KUKA KRL program: f1_Kuka_APT227T02S27.SRC

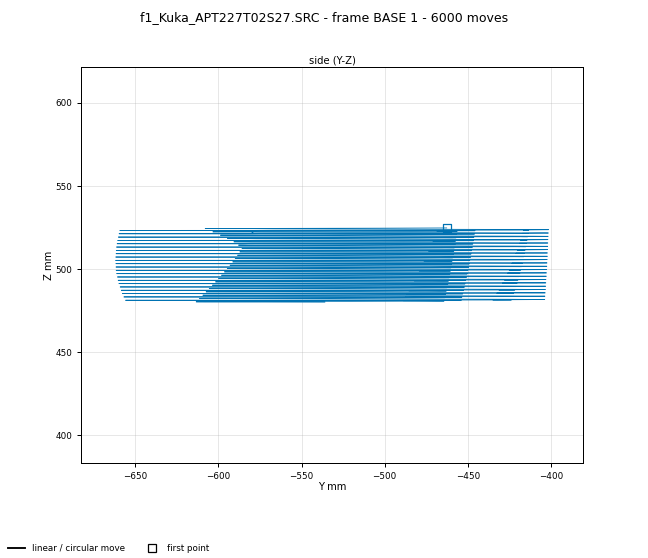
[picture p0: tool path of f1_Kuka_APT227T02S27.SRC in frame BASE 1, 6000 of 6001 moves have a stored position in this frame; points joined in program order, loops and branches not executed]
&ACCESS RVP
&REL 2
&PARAM TEMPLATE = C:\KRC\Roboter\Template\vorgabe
&PARAM EDITMASK = *
DEF f1_Kuka_APT227T02S27()


;FOLD INI;%{PE}%V3.2.0,%MKUKATPBASIS,%CINIT,%VCOMMON,%P
  ;FOLD BAS INI;%{E}%V3.2.0,%MKUKATPBASIS,%CINIT,%VINIT,%P
    GLOBAL INTERRUPT DECL 3 WHEN $STOPMESS==TRUE DO IR_STOPM ( )
    INTERRUPT ON 3
    BAS (#INITMOV,0 )
  ;ENDFOLD (BAS INI)
  ;FOLD USER INI;%{E}%V3.2.0,%MKUKATPUSER,%CINIT,%VINIT,%P
    ;Make your modifications here
  ;ENDFOLD (USER INI)
;ENDFOLD (INI)


;*** Make Null PTP Move
  PTP $pos_act

;*** Auto Load The Correct TOOL Data
  $tool=tool_data[2]

;*** Auto Load The Correct BASE Data
  $base=base_data[1]

  $ADVANCE = 5

;*** Restate Last Velocity
MMPM(30000.0)
SetRPM(8000)
LIN {X -0.077,Y -462.721,Z 524.797,A 0.000,B 0.000,C 90.000,E1 359.484} C_DIS
LIN {X 0.049,Y -465.139,Z 524.785,A 0.000,B 0.000,C 90.000,E1 357.249} C_DIS
LIN {X 0.032,Y -467.419,Z 524.774,A 0.000,B 0.000,C 90.000,E1 355.355} C_DIS
LIN {X 0.101,Y -469.908,Z 524.764,A 0.000,B 0.000,C 90.000,E1 353.457} C_DIS
LIN {X 0.052,Y -472.073,Z 524.755,A 0.000,B 0.000,C 90.000,E1 351.894} C_DIS
LIN {X 0.050,Y -474.231,Z 524.746,A 0.000,B 0.000,C 90.000,E1 350.330} C_DIS
LIN {X 0.160,Y -477.861,Z 524.733,A 0.000,B 0.000,C 90.000,E1 347.825} C_DIS
LIN {X -0.205,Y -484.314,Z 524.712,A 0.000,B 0.000,C 90.000,E1 344.157} C_DIS
LIN {X -0.147,Y -488.007,Z 524.702,A 0.000,B 0.000,C 90.000,E1 342.308} C_DIS
LIN {X 0.164,Y -492.282,Z 524.690,A 0.000,B 0.000,C 90.000,E1 340.134} C_DIS
LIN {X -0.090,Y -495.401,Z 524.681,A 0.000,B 0.000,C 90.000,E1 338.646} C_DIS
LIN {X 0.247,Y -499.060,Z 524.671,A 0.000,B 0.000,C 90.000,E1 336.794} C_DIS
LIN {X -0.055,Y -502.521,Z 524.661,A 0.000,B 0.000,C 90.000,E1 335.025} C_DIS
LIN {X 0.090,Y -505.373,Z 524.653,A 0.000,B 0.000,C 90.000,E1 333.512} C_DIS
LIN {X 0.140,Y -508.743,Z 524.643,A 0.000,B 0.000,C 90.000,E1 331.719} C_DIS
LIN {X -0.036,Y -511.558,Z 524.635,A 0.000,B 0.000,C 90.000,E1 330.255} C_DIS
LIN {X 0.202,Y -514.898,Z 524.625,A 0.000,B 0.000,C 90.000,E1 328.456} C_DIS
LIN {X 0.138,Y -517.811,Z 524.617,A 0.000,B 0.000,C 90.000,E1 326.993} C_DIS
LIN {X -0.035,Y -520.700,Z 524.609,A 0.000,B 0.000,C 90.000,E1 325.548} C_DIS
LIN {X 0.140,Y -523.590,Z 524.601,A 0.000,B 0.000,C 90.000,E1 324.069} C_DIS
LIN {X -0.116,Y -527.585,Z 524.589,A 0.000,B 0.000,C 90.000,E1 322.065} C_DIS
LIN {X 0.087,Y -530.439,Z 524.581,A 0.000,B 0.000,C 90.000,E1 320.598} C_DIS
LIN {X 0.267,Y -533.934,Z 524.572,A 0.000,B 0.000,C 90.000,E1 318.852} C_DIS
LIN {X 0.123,Y -538.133,Z 524.560,A 0.000,B 0.000,C 90.000,E1 316.863} C_DIS
LIN {X 0.048,Y -542.226,Z 524.549,A 0.000,B 0.000,C 90.000,E1 314.879} C_DIS
LIN {X 0.075,Y -546.335,Z 524.538,A 0.000,B 0.000,C 90.000,E1 312.894} C_DIS
LIN {X -0.075,Y -552.002,Z 524.524,A 0.000,B 0.000,C 90.000,E1 310.378} C_DIS
LIN {X -0.188,Y -555.087,Z 524.517,A 0.000,B 0.000,C 90.000,E1 308.991} C_DIS
LIN {X -0.057,Y -556.853,Z 524.512,A 0.000,B 0.000,C 90.000,E1 308.141} C_DIS
LIN {X 0.202,Y -560.643,Z 524.501,A 0.000,B 0.000,C 90.000,E1 306.171} C_DIS
LIN {X -0.099,Y -564.900,Z 524.491,A 0.000,B 0.000,C 90.000,E1 304.405} C_DIS
LIN {X -0.058,Y -566.045,Z 524.489,A 0.000,B 0.000,C 90.000,E1 304.072} C_DIS
LIN {X -0.050,Y -567.206,Z 524.487,A 0.000,B 0.000,C 90.000,E1 303.658} C_DIS
LIN {X -0.322,Y -568.426,Z 524.485,A 0.000,B 0.000,C 90.000,E1 303.372} C_DIS
LIN {X -0.206,Y -569.355,Z 524.484,A 0.000,B 0.000,C 90.000,E1 303.086} C_DIS
LIN {X -0.048,Y -571.821,Z 524.481,A 0.000,B 0.000,C 90.000,E1 302.625} C_DIS
LIN {X 0.075,Y -573.184,Z 524.480,A 0.000,B 0.000,C 90.000,E1 302.339} C_DIS
LIN {X 0.181,Y -575.458,Z 524.478,A 0.000,B 0.000,C 90.000,E1 301.926} C_DIS
LIN {X 0.020,Y -576.825,Z 524.476,A 0.000,B 0.000,C 90.000,E1 301.750} C_DIS
LIN {X 0.006,Y -580.151,Z 524.473,A 0.000,B 0.000,C 90.000,E1 301.209} C_DIS
LIN {X -0.052,Y -584.614,Z 524.470,A 0.000,B 0.000,C 90.000,E1 300.541} C_DIS
LIN {X -0.076,Y -589.187,Z 524.466,A 0.000,B 0.000,C 90.000,E1 299.873} C_DIS
LIN {X 0.186,Y -591.789,Z 524.464,A 0.000,B 0.000,C 90.000,E1 299.461} C_DIS
LIN {X -0.159,Y -597.723,Z 524.459,A 0.000,B 0.000,C 90.000,E1 298.565} C_DIS
LIN {X -0.113,Y -602.317,Z 524.454,A 0.000,B 0.000,C 90.000,E1 297.769} C_DIS
LIN {X -0.182,Y -603.762,Z 524.453,A 0.000,B 0.000,C 90.000,E1 297.513} C_DIS
LIN {X 0.179,Y -606.777,Z 524.448,A 0.000,B 0.000,C 90.000,E1 296.693} C_DIS
LIN {X 0.127,Y -607.269,Z 524.447,A 0.000,B 0.000,C 90.000,E1 296.437} C_DIS
LIN {X 0.031,Y -607.988,Z 524.444,A 0.000,B 0.000,C 90.000,E1 295.924} C_DIS
LIN {X -0.061,Y -607.894,Z 524.441,A 0.000,B 0.000,C 90.000,E1 295.412} C_DIS
LIN {X -0.108,Y -607.568,Z 524.440,A 0.000,B 0.000,C 90.000,E1 295.155} C_DIS
LIN {X -0.202,Y -606.152,Z 524.437,A 0.000,B 0.000,C 90.000,E1 294.643} C_DIS
LIN {X -0.229,Y -605.450,Z 524.436,A 0.000,B 0.000,C 90.000,E1 294.515} C_DIS
LIN {X 0.208,Y -601.708,Z 524.433,A 0.000,B 0.000,C 90.000,E1 293.951} C_DIS
LIN {X 0.191,Y -598.931,Z 524.432,A 0.000,B 0.000,C 90.000,E1 293.695} C_DIS
LIN {X 0.140,Y -595.749,Z 524.430,A 0.000,B 0.000,C 90.000,E1 293.462} C_DIS
LIN {X 0.124,Y -590.658,Z 524.429,A 0.000,B 0.000,C 90.000,E1 293.153} C_DIS
LIN {X -0.082,Y -583.314,Z 524.426,A 0.000,B 0.000,C 90.000,E1 292.717} C_DIS
LIN {X 0.230,Y -582.290,Z 524.426,A 0.000,B 0.000,C 90.000,E1 292.589} C_DIS
LIN {X 0.249,Y -580.640,Z 524.425,A 0.000,B 0.000,C 90.000,E1 292.461} C_DIS
LIN {X 0.267,Y -579.791,Z 524.424,A 0.000,B 0.000,C 90.000,E1 292.333} C_DIS
LIN {X 0.195,Y -579.183,Z 524.424,A 0.000,B 0.000,C 90.000,E1 292.206} C_DIS
LIN {X -0.313,Y -578.283,Z 524.421,A 0.000,B 0.000,C 90.000,E1 291.844} C_DIS
LIN {X -0.004,Y -578.140,Z 524.419,A 0.000,B 0.000,C 90.000,E1 291.408} C_DIS
LIN {X 0.269,Y -578.694,Z 524.410,A 0.000,B 0.000,C 90.000,E1 289.758} C_DIS
LIN {X -0.219,Y -578.876,Z 524.404,A 0.000,B 0.000,C 90.000,E1 288.725} C_DIS
LIN {X 0.047,Y -578.912,Z 524.396,A 0.000,B 0.000,C 90.000,E1 287.347} C_DIS
LIN {X 0.107,Y -578.758,Z 524.390,A 0.000,B 0.000,C 90.000,E1 286.260} C_DIS
LIN {X -0.133,Y -578.314,Z 524.381,A 0.000,B 0.000,C 90.000,E1 284.662} C_DIS
LIN {X -0.250,Y -578.005,Z 524.375,A 0.000,B 0.000,C 90.000,E1 283.592} C_DIS
LIN {X -0.292,Y -577.573,Z 524.368,A 0.000,B 0.000,C 90.000,E1 282.243} C_DIS
LIN {X -0.129,Y -576.982,Z 524.359,A 0.000,B 0.000,C 90.000,E1 280.602} C_DIS
LIN {X -0.094,Y -576.379,Z 524.350,A 0.000,B 0.000,C 90.000,E1 278.973} C_DIS
LIN {X -0.034,Y -575.668,Z 524.339,A 0.000,B 0.000,C 90.000,E1 277.068} C_DIS
LIN {X -0.073,Y -575.376,Z 524.335,A 0.000,B 0.000,C 90.000,E1 276.258} C_DIS
LIN {X 0.152,Y -574.823,Z 524.327,A 0.000,B 0.000,C 90.000,E1 274.878} C_DIS
LIN {X -0.206,Y -574.085,Z 524.320,A 0.000,B 0.000,C 90.000,E1 273.555} C_DIS
LIN {X -0.041,Y -573.161,Z 524.312,A 0.000,B 0.000,C 90.000,E1 272.178} C_DIS
LIN {X 0.244,Y -571.924,Z 524.303,A 0.000,B 0.000,C 90.000,E1 270.516} C_DIS
LIN {X -0.084,Y -570.447,Z 524.294,A 0.000,B 0.000,C 90.000,E1 268.912} C_DIS
LIN {X 0.012,Y -569.173,Z 524.286,A 0.000,B 0.000,C 90.000,E1 267.535} C_DIS
LIN {X -0.033,Y -568.111,Z 524.280,A 0.000,B 0.000,C 90.000,E1 266.445} C_DIS
LIN {X -0.098,Y -567.114,Z 524.274,A 0.000,B 0.000,C 90.000,E1 265.355} C_DIS
LIN {X 0.029,Y -565.712,Z 524.267,A 0.000,B 0.000,C 90.000,E1 263.970} C_DIS
LIN {X -0.019,Y -564.454,Z 524.260,A 0.000,B 0.000,C 90.000,E1 262.875} C_DIS
LIN {X 0.066,Y -562.811,Z 524.253,A 0.000,B 0.000,C 90.000,E1 261.489} C_DIS
LIN {X -0.046,Y -560.309,Z 524.242,A 0.000,B 0.000,C 90.000,E1 259.567} C_DIS
LIN {X 0.183,Y -558.097,Z 524.233,A 0.000,B 0.000,C 90.000,E1 257.881} C_DIS
LIN {X 0.193,Y -556.461,Z 524.227,A 0.000,B 0.000,C 90.000,E1 256.769} C_DIS
LIN {X -0.231,Y -554.729,Z 524.220,A 0.000,B 0.000,C 90.000,E1 255.700} C_DIS
LIN {X -0.021,Y -552.386,Z 524.213,A 0.000,B 0.000,C 90.000,E1 254.283} C_DIS
LIN {X -0.238,Y -549.770,Z 524.205,A 0.000,B 0.000,C 90.000,E1 252.906} C_DIS
LIN {X 0.189,Y -546.847,Z 524.197,A 0.000,B 0.000,C 90.000,E1 251.456} C_DIS
LIN {X -0.198,Y -544.424,Z 524.191,A 0.000,B 0.000,C 90.000,E1 250.369} C_DIS
LIN {X -0.195,Y -541.220,Z 524.183,A 0.000,B 0.000,C 90.000,E1 248.954} C_DIS
LIN {X 0.028,Y -538.498,Z 524.177,A 0.000,B 0.000,C 90.000,E1 247.794} C_DIS
LIN {X -0.085,Y -535.669,Z 524.170,A 0.000,B 0.000,C 90.000,E1 246.666} C_DIS
LIN {X 0.251,Y -532.662,Z 524.164,A 0.000,B 0.000,C 90.000,E1 245.485} C_DIS
LIN {X -0.015,Y -528.732,Z 524.156,A 0.000,B 0.000,C 90.000,E1 244.076} C_DIS
LIN {X -0.035,Y -525.449,Z 524.150,A 0.000,B 0.000,C 90.000,E1 242.922} C_DIS
LIN {X -0.038,Y -520.512,Z 524.140,A 0.000,B 0.000,C 90.000,E1 241.179} C_DIS
LIN {X 0.090,Y -515.420,Z 524.130,A 0.000,B 0.000,C 90.000,E1 239.410} C_DIS
LIN {X -0.068,Y -511.862,Z 524.124,A 0.000,B 0.000,C 90.000,E1 238.250} C_DIS
LIN {X -0.313,Y -506.357,Z 524.114,A 0.000,B 0.000,C 90.000,E1 236.501} C_DIS
LIN {X -0.084,Y -498.136,Z 524.099,A 0.000,B 0.000,C 90.000,E1 233.783} C_DIS
LIN {X -0.034,Y -492.194,Z 524.087,A 0.000,B 0.000,C 90.000,E1 231.662} C_DIS
LIN {X 0.033,Y -487.110,Z 524.077,A 0.000,B 0.000,C 90.000,E1 229.828} C_DIS
LIN {X 0.056,Y -481.384,Z 524.065,A 0.000,B 0.000,C 90.000,E1 227.676} C_DIS
LIN {X 0.112,Y -479.029,Z 524.060,A 0.000,B 0.000,C 90.000,E1 226.743} C_DIS
LIN {X -0.205,Y -474.304,Z 524.049,A 0.000,B 0.000,C 90.000,E1 224.919} C_DIS
LIN {X 0.190,Y -471.260,Z 524.043,A 0.000,B 0.000,C 90.000,E1 223.623} C_DIS
LIN {X 0.039,Y -466.719,Z 524.032,A 0.000,B 0.000,C 90.000,E1 221.757} C_DIS
LIN {X 0.083,Y -463.152,Z 524.023,A 0.000,B 0.000,C 90.000,E1 220.172} C_DIS
LIN {X 0.155,Y -458.881,Z 524.013,A 0.000,B 0.000,C 90.000,E1 218.257} C_DIS
LIN {X 0.118,Y -455.424,Z 524.004,A 0.000,B 0.000,C 90.000,E1 216.664} C_DIS
LIN {X -0.116,Y -450.036,Z 523.990,A 0.000,B 0.000,C 90.000,E1 214.119} C_DIS
LIN {X 0.278,Y -445.614,Z 523.977,A 0.000,B 0.000,C 90.000,E1 211.799} C_DIS
LIN {X 0.084,Y -441.282,Z 523.964,A 0.000,B 0.000,C 90.000,E1 209.539} C_DIS
LIN {X 0.086,Y -438.420,Z 523.955,A 0.000,B 0.000,C 90.000,E1 207.897} C_DIS
LIN {X 0.037,Y -434.989,Z 523.944,A 0.000,B 0.000,C 90.000,E1 205.924} C_DIS
LIN {X 0.124,Y -431.091,Z 523.931,A 0.000,B 0.000,C 90.000,E1 203.590} C_DIS
LIN {X -0.074,Y -426.498,Z 523.914,A 0.000,B 0.000,C 90.000,E1 200.610} C_DIS
LIN {X -0.109,Y -423.681,Z 523.903,A 0.000,B 0.000,C 90.000,E1 198.598} C_DIS
LIN {X 0.106,Y -420.675,Z 523.890,A 0.000,B 0.000,C 90.000,E1 196.205} C_DIS
LIN {X 0.071,Y -418.208,Z 523.879,A 0.000,B 0.000,C 90.000,E1 194.175} C_DIS
LIN {X -0.141,Y -414.972,Z 523.864,A 0.000,B 0.000,C 90.000,E1 191.478} C_DIS
LIN {X 0.201,Y -412.776,Z 523.852,A 0.000,B 0.000,C 90.000,E1 189.378} C_DIS
LIN {X -0.085,Y -410.985,Z 523.843,A 0.000,B 0.000,C 90.000,E1 187.701} C_DIS
LIN {X -0.004,Y -408.416,Z 523.829,A 0.000,B 0.000,C 90.000,E1 185.277} C_DIS
LIN {X -0.157,Y -405.178,Z 523.808,A 0.000,B 0.000,C 90.000,E1 181.489} C_DIS
LIN {X 0.111,Y -404.005,Z 523.799,A 0.000,B 0.000,C 90.000,E1 179.714} C_DIS
LIN {X 0.196,Y -402.337,Z 523.779,A 0.000,B 0.000,C 90.000,E1 176.216} C_DIS
LIN {X -0.068,Y -401.559,Z 523.760,A 0.000,B 0.000,C 90.000,E1 172.761} C_DIS
LIN {X -0.180,Y -401.451,Z 523.746,A 0.000,B 0.000,C 90.000,E1 170.330} C_DIS
LIN {X -0.163,Y -401.675,Z 523.733,A 0.000,B 0.000,C 90.000,E1 167.881} C_DIS
LIN {X 0.118,Y -402.370,Z 523.717,A 0.000,B 0.000,C 90.000,E1 165.046} C_DIS
LIN {X -0.152,Y -403.611,Z 523.700,A 0.000,B 0.000,C 90.000,E1 161.945} C_DIS
LIN {X -0.219,Y -404.872,Z 523.686,A 0.000,B 0.000,C 90.000,E1 159.518} C_DIS
LIN {X -0.062,Y -406.219,Z 523.674,A 0.000,B 0.000,C 90.000,E1 157.411} C_DIS
LIN {X 0.025,Y -407.955,Z 523.661,A 0.000,B 0.000,C 90.000,E1 154.973} C_DIS
LIN {X -0.056,Y -409.262,Z 523.651,A 0.000,B 0.000,C 90.000,E1 153.256} C_DIS
LIN {X 0.148,Y -410.253,Z 523.644,A 0.000,B 0.000,C 90.000,E1 151.847} C_DIS
LIN {X 0.130,Y -411.453,Z 523.634,A 0.000,B 0.000,C 90.000,E1 150.127} C_DIS
LIN {X 0.136,Y -412.492,Z 523.625,A 0.000,B 0.000,C 90.000,E1 148.408} C_DIS
LIN {X 0.023,Y -413.428,Z 523.615,A 0.000,B 0.000,C 90.000,E1 146.707} C_DIS
LIN {X 0.089,Y -414.386,Z 523.604,A 0.000,B 0.000,C 90.000,E1 144.642} C_DIS
LIN {X -0.036,Y -414.932,Z 523.596,A 0.000,B 0.000,C 90.000,E1 143.290} C_DIS
LIN {X -0.080,Y -415.302,Z 523.590,A 0.000,B 0.000,C 90.000,E1 142.271} C_DIS
LIN {X -0.073,Y -415.857,Z 523.581,A 0.000,B 0.000,C 90.000,E1 140.561} C_DIS
LIN {X 0.076,Y -416.211,Z 523.573,A 0.000,B 0.000,C 90.000,E1 139.175} C_DIS
LIN {X -0.127,Y -416.501,Z 523.566,A 0.000,B 0.000,C 90.000,E1 137.838} C_DIS
LIN {X -0.139,Y -416.692,Z 523.556,A 0.000,B 0.000,C 90.000,E1 136.134} C_DIS
LIN {X -0.163,Y -416.692,Z 523.547,A 0.000,B 0.000,C 90.000,E1 134.433} C_DIS
LIN {X -0.067,Y -416.630,Z 523.539,A 0.000,B 0.000,C 90.000,E1 133.056} C_DIS
LIN {X 0.043,Y -416.317,Z 523.532,A 0.000,B 0.000,C 90.000,E1 131.676} C_DIS
LIN {X -0.121,Y -415.764,Z 523.524,A 0.000,B 0.000,C 90.000,E1 130.334} C_DIS
LIN {X -0.028,Y -414.918,Z 523.516,A 0.000,B 0.000,C 90.000,E1 128.955} C_DIS
LIN {X 0.204,Y -413.541,Z 523.505,A 0.000,B 0.000,C 90.000,E1 126.870} C_DIS
LIN {X 0.071,Y -413.402,Z 523.504,A 0.000,B 0.000,C 90.000,E1 126.664} C_DIS
LIN {X 0.032,Y -413.404,Z 523.504,A 0.000,B 0.000,C 90.000,E1 126.664} C_DIS
LIN {X -0.101,Y -415.792,Z 523.499,A 0.000,B 0.000,C 90.000,E1 125.884} C_DIS
LIN {X 0.006,Y -425.244,Z 523.479,A 0.000,B 0.000,C 90.000,E1 122.133} C_DIS
LIN {X -0.061,Y -430.248,Z 523.469,A 0.000,B 0.000,C 90.000,E1 120.463} C_DIS
LIN {X -0.062,Y -431.151,Z 523.467,A 0.000,B 0.000,C 90.000,E1 120.129} C_DIS
LIN {X -0.117,Y -440.260,Z 523.447,A 0.000,B 0.000,C 90.000,E1 116.488} C_DIS
LIN {X 0.076,Y -445.002,Z 523.438,A 0.000,B 0.000,C 90.000,E1 114.823} C_DIS
LIN {X -0.016,Y -453.050,Z 523.419,A 0.000,B 0.000,C 90.000,E1 111.354} C_DIS
LIN {X -0.056,Y -453.112,Z 523.419,A 0.000,B 0.000,C 90.000,E1 111.354} C_DIS
LIN {X 0.157,Y -476.770,Z 523.414,A 0.000,B 0.000,C 90.000,E1 110.482} C_DIS
LIN {X -0.054,Y -494.356,Z 523.410,A 0.000,B 0.000,C 90.000,E1 109.885} C_DIS
LIN {X -0.133,Y -504.552,Z 523.408,A 0.000,B 0.000,C 90.000,E1 109.504} C_DIS
LIN {X -0.077,Y -514.947,Z 523.406,A 0.000,B 0.000,C 90.000,E1 109.087} C_DIS
LIN {X -0.100,Y -526.904,Z 523.403,A 0.000,B 0.000,C 90.000,E1 108.598} C_DIS
LIN {X -0.099,Y -535.317,Z 523.401,A 0.000,B 0.000,C 90.000,E1 108.236} C_DIS
LIN {X -0.030,Y -545.219,Z 523.399,A 0.000,B 0.000,C 90.000,E1 107.764} C_DIS
LIN {X 0.036,Y -552.939,Z 523.396,A 0.000,B 0.000,C 90.000,E1 107.330} C_DIS
LIN {X 0.190,Y -557.612,Z 523.395,A 0.000,B 0.000,C 90.000,E1 107.040} C_DIS
LIN {X -0.112,Y -563.564,Z 523.393,A 0.000,B 0.000,C 90.000,E1 106.677} C_DIS
LIN {X 0.322,Y -567.952,Z 523.391,A 0.000,B 0.000,C 90.000,E1 106.315} C_DIS
LIN {X -0.104,Y -575.047,Z 523.388,A 0.000,B 0.000,C 90.000,E1 105.788} C_DIS
LIN {X -0.054,Y -580.373,Z 523.385,A 0.000,B 0.000,C 90.000,E1 105.300} C_DIS
LIN {X 0.038,Y -585.188,Z 523.382,A 0.000,B 0.000,C 90.000,E1 104.828} C_DIS
LIN {X -0.325,Y -588.649,Z 523.380,A 0.000,B 0.000,C 90.000,E1 104.481} C_DIS
LIN {X 0.157,Y -589.982,Z 523.380,A 0.000,B 0.000,C 90.000,E1 104.300} C_DIS
LIN {X 0.082,Y -595.263,Z 523.376,A 0.000,B 0.000,C 90.000,E1 103.703} C_DIS
LIN {X 0.209,Y -601.269,Z 523.372,A 0.000,B 0.000,C 90.000,E1 102.939} C_DIS
LIN {X 0.282,Y -606.103,Z 523.369,A 0.000,B 0.000,C 90.000,E1 102.299} C_DIS
LIN {X 0.088,Y -611.856,Z 523.364,A 0.000,B 0.000,C 90.000,E1 101.535} C_DIS
LIN {X 0.119,Y -616.974,Z 523.360,A 0.000,B 0.000,C 90.000,E1 100.782} C_DIS
LIN {X -0.141,Y -622.460,Z 523.355,A 0.000,B 0.000,C 90.000,E1 99.905} C_DIS
LIN {X -0.134,Y -626.099,Z 523.351,A 0.000,B 0.000,C 90.000,E1 99.265} C_DIS
LIN {X -0.097,Y -629.550,Z 523.348,A 0.000,B 0.000,C 90.000,E1 98.624} C_DIS
LIN {X -0.154,Y -633.941,Z 523.343,A 0.000,B 0.000,C 90.000,E1 97.757} C_DIS
LIN {X -0.199,Y -637.640,Z 523.339,A 0.000,B 0.000,C 90.000,E1 97.004} C_DIS
LIN {X 0.166,Y -642.290,Z 523.333,A 0.000,B 0.000,C 90.000,E1 95.967} C_DIS
LIN {X 0.129,Y -645.562,Z 523.329,A 0.000,B 0.000,C 90.000,E1 95.220} C_DIS
LIN {X 0.127,Y -648.555,Z 523.325,A 0.000,B 0.000,C 90.000,E1 94.473} C_DIS
LIN {X 0.157,Y -651.236,Z 523.321,A 0.000,B 0.000,C 90.000,E1 93.726} C_DIS
LIN {X -0.059,Y -652.132,Z 523.319,A 0.000,B 0.000,C 90.000,E1 93.498} C_DIS
LIN {X 0.004,Y -654.338,Z 523.315,A 0.000,B 0.000,C 90.000,E1 92.751} C_DIS
LIN {X 0.256,Y -655.673,Z 523.313,A 0.000,B 0.000,C 90.000,E1 92.236} C_DIS
LIN {X -0.115,Y -656.783,Z 523.310,A 0.000,B 0.000,C 90.000,E1 91.776} C_DIS
LIN {X 0.156,Y -657.700,Z 523.307,A 0.000,B 0.000,C 90.000,E1 91.260} C_DIS
LIN {X 0.248,Y -658.652,Z 523.303,A 0.000,B 0.000,C 90.000,E1 90.516} C_DIS
LIN {X -0.122,Y -659.068,Z 523.300,A 0.000,B 0.000,C 90.000,E1 90.057} C_DIS
LIN {X 0.169,Y -659.308,Z 523.298,A 0.000,B 0.000,C 90.000,E1 89.542} C_DIS
LIN {X 0.278,Y -659.279,Z 523.294,A 0.000,B 0.000,C 90.000,E1 88.797} C_DIS
LIN {X -0.091,Y -659.081,Z 523.291,A 0.000,B 0.000,C 90.000,E1 88.339} C_DIS
LIN {X 0.034,Y -658.396,Z 523.287,A 0.000,B 0.000,C 90.000,E1 87.593} C_DIS
LIN {X -0.153,Y -658.166,Z 523.285,A 0.000,B 0.000,C 90.000,E1 87.364} C_DIS
LIN {X -0.030,Y -656.998,Z 523.281,A 0.000,B 0.000,C 90.000,E1 86.617} C_DIS
LIN {X 0.237,Y -656.103,Z 523.279,A 0.000,B 0.000,C 90.000,E1 86.102} C_DIS
LIN {X -0.114,Y -655.018,Z 523.276,A 0.000,B 0.000,C 90.000,E1 85.641} C_DIS
LIN {X -0.020,Y -653.077,Z 523.272,A 0.000,B 0.000,C 90.000,E1 84.894} C_DIS
LIN {X -0.101,Y -650.007,Z 523.266,A 0.000,B 0.000,C 90.000,E1 83.913} C_DIS
LIN {X -0.062,Y -647.376,Z 523.262,A 0.000,B 0.000,C 90.000,E1 83.166} C_DIS
LIN {X -0.219,Y -643.396,Z 523.257,A 0.000,B 0.000,C 90.000,E1 82.186} C_DIS
LIN {X -0.170,Y -640.058,Z 523.252,A 0.000,B 0.000,C 90.000,E1 81.432} C_DIS
LIN {X -0.015,Y -637.052,Z 523.249,A 0.000,B 0.000,C 90.000,E1 80.792} C_DIS
LIN {X 0.114,Y -633.781,Z 523.245,A 0.000,B 0.000,C 90.000,E1 80.151} C_DIS
LIN {X -0.096,Y -628.841,Z 523.240,A 0.000,B 0.000,C 90.000,E1 79.285} C_DIS
LIN {X 0.283,Y -626.571,Z 523.238,A 0.000,B 0.000,C 90.000,E1 78.870} C_DIS
LIN {X 0.148,Y -621.784,Z 523.234,A 0.000,B 0.000,C 90.000,E1 78.117} C_DIS
LIN {X -0.289,Y -618.585,Z 523.231,A 0.000,B 0.000,C 90.000,E1 77.645} C_DIS
LIN {X 0.137,Y -613.548,Z 523.227,A 0.000,B 0.000,C 90.000,E1 76.881} C_DIS
LIN {X 0.135,Y -607.509,Z 523.223,A 0.000,B 0.000,C 90.000,E1 76.117} C_DIS
LIN {X 0.201,Y -602.910,Z 523.220,A 0.000,B 0.000,C 90.000,E1 75.589} C_DIS
LIN {X -0.023,Y -598.092,Z 523.217,A 0.000,B 0.000,C 90.000,E1 75.102} C_DIS
LIN {X -0.254,Y -591.907,Z 523.214,A 0.000,B 0.000,C 90.000,E1 74.519} C_DIS
LIN {X 0.284,Y -586.401,Z 523.211,A 0.000,B 0.000,C 90.000,E1 73.976} C_DIS
LIN {X -0.192,Y -580.627,Z 523.209,A 0.000,B 0.000,C 90.000,E1 73.559} C_DIS
LIN {X -0.270,Y -574.898,Z 523.206,A 0.000,B 0.000,C 90.000,E1 73.142} C_DIS
LIN {X 0.184,Y -570.285,Z 523.204,A 0.000,B 0.000,C 90.000,E1 72.779} C_DIS
LIN {X 0.244,Y -563.718,Z 523.202,A 0.000,B 0.000,C 90.000,E1 72.362} C_DIS
LIN {X -0.177,Y -558.688,Z 523.201,A 0.000,B 0.000,C 90.000,E1 72.127} C_DIS
LIN {X -0.186,Y -553.667,Z 523.199,A 0.000,B 0.000,C 90.000,E1 71.873} C_DIS
LIN {X 0.090,Y -546.412,Z 523.198,A 0.000,B 0.000,C 90.000,E1 71.529} C_DIS
LIN {X -0.015,Y -540.962,Z 523.196,A 0.000,B 0.000,C 90.000,E1 71.329} C_DIS
LIN {X -0.084,Y -535.612,Z 523.195,A 0.000,B 0.000,C 90.000,E1 71.148} C_DIS
LIN {X 0.021,Y -527.801,Z 523.194,A 0.000,B 0.000,C 90.000,E1 70.913} C_DIS
LIN {X -0.208,Y -514.834,Z 523.192,A 0.000,B 0.000,C 90.000,E1 70.604} C_DIS
LIN {X 0.078,Y -503.831,Z 523.191,A 0.000,B 0.000,C 90.000,E1 70.315} C_DIS
LIN {X 0.160,Y -494.116,Z 523.190,A 0.000,B 0.000,C 90.000,E1 70.115} C_DIS
LIN {X -0.070,Y -483.073,Z 523.189,A 0.000,B 0.000,C 90.000,E1 69.934} C_DIS
LIN {X -0.068,Y -469.667,Z 523.187,A 0.000,B 0.000,C 90.000,E1 69.699} C_DIS
LIN {X -0.102,Y -469.642,Z 523.187,A 0.000,B 0.000,C 90.000,E1 69.699} C_DIS
LIN {X -0.100,Y -465.762,Z 523.173,A 0.000,B 0.000,C 90.000,E1 67.155} C_DIS
LIN {X 0.144,Y -463.664,Z 523.168,A 0.000,B 0.000,C 90.000,E1 66.177} C_DIS
LIN {X 0.230,Y -455.727,Z 523.145,A 0.000,B 0.000,C 90.000,E1 62.025} C_DIS
LIN {X 0.119,Y -455.083,Z 523.143,A 0.000,B 0.000,C 90.000,E1 61.719} C_DIS
LIN {X -0.054,Y -446.436,Z 523.122,A 0.000,B 0.000,C 90.000,E1 57.867} C_DIS
LIN {X 0.076,Y -445.686,Z 523.119,A 0.000,B 0.000,C 90.000,E1 57.454} C_DIS
LIN {X 0.036,Y -445.699,Z 523.119,A 0.000,B 0.000,C 90.000,E1 57.454} C_DIS
LIN {X 0.223,Y -450.097,Z 523.111,A 0.000,B 0.000,C 90.000,E1 55.881} C_DIS
LIN {X -0.288,Y -452.595,Z 523.105,A 0.000,B 0.000,C 90.000,E1 54.975} C_DIS
LIN {X -0.060,Y -456.379,Z 523.096,A 0.000,B 0.000,C 90.000,E1 53.336} C_DIS
LIN {X 0.037,Y -457.767,Z 523.093,A 0.000,B 0.000,C 90.000,E1 52.683} C_DIS
LIN {X -0.118,Y -459.541,Z 523.087,A 0.000,B 0.000,C 90.000,E1 51.743} C_DIS
LIN {X -0.127,Y -462.114,Z 523.079,A 0.000,B 0.000,C 90.000,E1 50.150} C_DIS
LIN {X 0.102,Y -463.873,Z 523.072,A 0.000,B 0.000,C 90.000,E1 48.852} C_DIS
LIN {X -0.044,Y -465.024,Z 523.066,A 0.000,B 0.000,C 90.000,E1 47.919} C_DIS
LIN {X -0.174,Y -466.013,Z 523.061,A 0.000,B 0.000,C 90.000,E1 46.986} C_DIS
LIN {X -0.295,Y -466.818,Z 523.056,A 0.000,B 0.000,C 90.000,E1 46.053} C_DIS
LIN {X -0.084,Y -467.481,Z 523.050,A 0.000,B 0.000,C 90.000,E1 45.081} C_DIS
LIN {X 0.137,Y -468.036,Z 523.045,A 0.000,B 0.000,C 90.000,E1 44.109} C_DIS
LIN {X 0.114,Y -468.446,Z 523.038,A 0.000,B 0.000,C 90.000,E1 42.852} C_DIS
LIN {X 0.095,Y -468.615,Z 523.031,A 0.000,B 0.000,C 90.000,E1 41.595} C_DIS
LIN {X 0.119,Y -468.463,Z 523.024,A 0.000,B 0.000,C 90.000,E1 40.334} C_DIS
LIN {X -0.216,Y -468.162,Z 523.017,A 0.000,B 0.000,C 90.000,E1 39.116} C_DIS
LIN {X -0.016,Y -467.483,Z 523.007,A 0.000,B 0.000,C 90.000,E1 37.202} C_DIS
LIN {X 0.215,Y -466.709,Z 522.998,A 0.000,B 0.000,C 90.000,E1 35.598} C_DIS
LIN {X 0.051,Y -465.881,Z 522.989,A 0.000,B 0.000,C 90.000,E1 34.040} C_DIS
LIN {X -0.007,Y -464.940,Z 522.980,A 0.000,B 0.000,C 90.000,E1 32.467} C_DIS
LIN {X 0.068,Y -464.002,Z 522.972,A 0.000,B 0.000,C 90.000,E1 30.875} C_DIS
LIN {X -0.138,Y -462.740,Z 522.961,A 0.000,B 0.000,C 90.000,E1 28.999} C_DIS
LIN {X -0.010,Y -461.464,Z 522.951,A 0.000,B 0.000,C 90.000,E1 27.078} C_DIS
LIN {X 0.014,Y -460.040,Z 522.938,A 0.000,B 0.000,C 90.000,E1 24.847} C_DIS
LIN {X -0.114,Y -459.033,Z 522.927,A 0.000,B 0.000,C 90.000,E1 22.950} C_DIS
LIN {X 0.050,Y -457.942,Z 522.913,A 0.000,B 0.000,C 90.000,E1 20.375} C_DIS
LIN {X -0.070,Y -457.267,Z 522.903,A 0.000,B 0.000,C 90.000,E1 18.471} C_DIS
LIN {X -0.208,Y -456.570,Z 522.887,A 0.000,B 0.000,C 90.000,E1 15.607} C_DIS
LIN {X -0.045,Y -456.427,Z 522.871,A 0.000,B 0.000,C 90.000,E1 12.703} C_DIS
LIN {X -0.056,Y -456.664,Z 522.860,A 0.000,B 0.000,C 90.000,E1 10.782} C_DIS
LIN {X 0.175,Y -457.228,Z 522.847,A 0.000,B 0.000,C 90.000,E1 8.511} C_DIS
LIN {X -0.173,Y -458.085,Z 522.835,A 0.000,B 0.000,C 90.000,E1 6.315} C_DIS
LIN {X 0.090,Y -459.503,Z 522.821,A 0.000,B 0.000,C 90.000,E1 3.726} C_DIS
LIN {X 0.138,Y -461.050,Z 522.808,A 0.000,B 0.000,C 90.000,E1 1.489} C_DIS
LIN {X -0.076,Y -462.867,Z 522.797,A 0.000,B 0.000,C 90.000,E1 359.484} C_DIS
LIN {X 0.054,Y -465.273,Z 522.785,A 0.000,B 0.000,C 90.000,E1 357.249} C_DIS
LIN {X 0.039,Y -467.544,Z 522.774,A 0.000,B 0.000,C 90.000,E1 355.355} C_DIS
LIN {X 0.111,Y -470.032,Z 522.764,A 0.000,B 0.000,C 90.000,E1 353.457} C_DIS
LIN {X -0.111,Y -472.621,Z 522.753,A 0.000,B 0.000,C 90.000,E1 351.602} C_DIS
LIN {X -0.103,Y -474.769,Z 522.745,A 0.000,B 0.000,C 90.000,E1 350.038} C_DIS
LIN {X 0.178,Y -477.984,Z 522.733,A 0.000,B 0.000,C 90.000,E1 347.825} C_DIS
LIN {X -0.041,Y -483.873,Z 522.714,A 0.000,B 0.000,C 90.000,E1 344.448} C_DIS
LIN {X -0.119,Y -488.161,Z 522.702,A 0.000,B 0.000,C 90.000,E1 342.308} C_DIS
LIN {X -0.264,Y -492.468,Z 522.690,A 0.000,B 0.000,C 90.000,E1 340.188} C_DIS
LIN {X -0.053,Y -495.579,Z 522.681,A 0.000,B 0.000,C 90.000,E1 338.646} C_DIS
LIN {X 0.226,Y -498.641,Z 522.673,A 0.000,B 0.000,C 90.000,E1 337.102} C_DIS
LIN {X 0.095,Y -501.572,Z 522.665,A 0.000,B 0.000,C 90.000,E1 335.613} C_DIS
LIN {X -0.237,Y -504.462,Z 522.656,A 0.000,B 0.000,C 90.000,E1 334.152} C_DIS
LIN {X -0.207,Y -507.868,Z 522.646,A 0.000,B 0.000,C 90.000,E1 332.359} C_DIS
LIN {X 0.131,Y -511.238,Z 522.636,A 0.000,B 0.000,C 90.000,E1 330.539} C_DIS
LIN {X -0.085,Y -514.653,Z 522.627,A 0.000,B 0.000,C 90.000,E1 328.791} C_DIS
LIN {X -0.223,Y -518.145,Z 522.617,A 0.000,B 0.000,C 90.000,E1 327.041} C_DIS
LIN {X 0.045,Y -521.037,Z 522.609,A 0.000,B 0.000,C 90.000,E1 325.548} C_DIS
LIN {X -0.197,Y -523.951,Z 522.601,A 0.000,B 0.000,C 90.000,E1 324.116} C_DIS
LIN {X 0.011,Y -527.420,Z 522.591,A 0.000,B 0.000,C 90.000,E1 322.351} C_DIS
LIN {X 0.213,Y -530.322,Z 522.583,A 0.000,B 0.000,C 90.000,E1 320.884} C_DIS
LIN {X 0.046,Y -533.791,Z 522.573,A 0.000,B 0.000,C 90.000,E1 319.175} C_DIS
LIN {X -0.093,Y -536.764,Z 522.565,A 0.000,B 0.000,C 90.000,E1 317.757} C_DIS
LIN {X -0.145,Y -539.195,Z 522.559,A 0.000,B 0.000,C 90.000,E1 316.620} C_DIS
LIN {X 0.191,Y -543.256,Z 522.548,A 0.000,B 0.000,C 90.000,E1 314.595} C_DIS
LIN {X -0.143,Y -546.692,Z 522.539,A 0.000,B 0.000,C 90.000,E1 312.933} C_DIS
LIN {X 0.091,Y -552.259,Z 522.524,A 0.000,B 0.000,C 90.000,E1 310.378} C_DIS
LIN {X -0.086,Y -554.742,Z 522.518,A 0.000,B 0.000,C 90.000,E1 309.277} C_DIS
LIN {X -0.225,Y -557.133,Z 522.512,A 0.000,B 0.000,C 90.000,E1 308.177} C_DIS
LIN {X 0.110,Y -559.275,Z 522.506,A 0.000,B 0.000,C 90.000,E1 307.030} C_DIS
LIN {X -0.016,Y -565.229,Z 522.490,A 0.000,B 0.000,C 90.000,E1 304.278} C_DIS
LIN {X 0.202,Y -566.732,Z 522.487,A 0.000,B 0.000,C 90.000,E1 303.706} C_DIS
LIN {X -0.001,Y -567.396,Z 522.486,A 0.000,B 0.000,C 90.000,E1 303.452} C_DIS
LIN {X 0.228,Y -569.107,Z 522.483,A 0.000,B 0.000,C 90.000,E1 302.880} C_DIS
LIN {X -0.011,Y -569.952,Z 522.482,A 0.000,B 0.000,C 90.000,E1 302.752} C_DIS
LIN {X 0.109,Y -571.087,Z 522.480,A 0.000,B 0.000,C 90.000,E1 302.467} C_DIS
LIN {X -0.076,Y -572.006,Z 522.479,A 0.000,B 0.000,C 90.000,E1 302.212} C_DIS
LIN {X 0.049,Y -573.384,Z 522.477,A 0.000,B 0.000,C 90.000,E1 301.926} C_DIS
LIN {X -0.038,Y -573.976,Z 522.477,A 0.000,B 0.000,C 90.000,E1 301.799} C_DIS
LIN {X -0.073,Y -576.985,Z 522.474,A 0.000,B 0.000,C 90.000,E1 301.258} C_DIS
LIN {X -0.014,Y -579.173,Z 522.471,A 0.000,B 0.000,C 90.000,E1 300.846} C_DIS
LIN {X 0.320,Y -588.155,Z 522.463,A 0.000,B 0.000,C 90.000,E1 299.333} C_DIS
LIN {X 0.121,Y -595.328,Z 522.457,A 0.000,B 0.000,C 90.000,E1 298.153} C_DIS
LIN {X -0.015,Y -597.485,Z 522.454,A 0.000,B 0.000,C 90.000,E1 297.769} C_DIS
LIN {X -0.220,Y -600.522,Z 522.451,A 0.000,B 0.000,C 90.000,E1 297.129} C_DIS
LIN {X -0.295,Y -601.462,Z 522.449,A 0.000,B 0.000,C 90.000,E1 296.873} C_DIS
LIN {X 0.106,Y -602.721,Z 522.446,A 0.000,B 0.000,C 90.000,E1 296.309} C_DIS
LIN {X 0.041,Y -603.162,Z 522.445,A 0.000,B 0.000,C 90.000,E1 296.052} C_DIS
LIN {X -0.022,Y -603.349,Z 522.443,A 0.000,B 0.000,C 90.000,E1 295.796} C_DIS
LIN {X -0.083,Y -603.390,Z 522.442,A 0.000,B 0.000,C 90.000,E1 295.540} C_DIS
LIN {X -0.205,Y -602.726,Z 522.439,A 0.000,B 0.000,C 90.000,E1 295.027} C_DIS
LIN {X -0.269,Y -602.259,Z 522.438,A 0.000,B 0.000,C 90.000,E1 294.771} C_DIS
LIN {X -0.301,Y -601.402,Z 522.437,A 0.000,B 0.000,C 90.000,E1 294.643} C_DIS
LIN {X 0.143,Y -599.371,Z 522.435,A 0.000,B 0.000,C 90.000,E1 294.207} C_DIS
LIN {X 0.107,Y -598.411,Z 522.434,A 0.000,B 0.000,C 90.000,E1 294.079} C_DIS
LIN {X 0.100,Y -594.628,Z 522.432,A 0.000,B 0.000,C 90.000,E1 293.695} C_DIS
LIN {X -0.225,Y -592.255,Z 522.431,A 0.000,B 0.000,C 90.000,E1 293.515} C_DIS
LIN {X 0.155,Y -587.306,Z 522.429,A 0.000,B 0.000,C 90.000,E1 293.131} C_DIS
LIN {X -0.058,Y -583.478,Z 522.427,A 0.000,B 0.000,C 90.000,E1 292.898} C_DIS
LIN {X -0.013,Y -581.170,Z 522.426,A 0.000,B 0.000,C 90.000,E1 292.642} C_DIS
LIN {X -0.228,Y -580.119,Z 522.425,A 0.000,B 0.000,C 90.000,E1 292.461} C_DIS
LIN {X -0.298,Y -579.673,Z 522.424,A 0.000,B 0.000,C 90.000,E1 292.333} C_DIS
LIN {X -0.135,Y -579.246,Z 522.422,A 0.000,B 0.000,C 90.000,E1 291.972} C_DIS
LIN {X 0.105,Y -579.080,Z 522.419,A 0.000,B 0.000,C 90.000,E1 291.408} C_DIS
LIN {X -0.146,Y -579.694,Z 522.410,A 0.000,B 0.000,C 90.000,E1 289.812} C_DIS
LIN {X -0.076,Y -579.922,Z 522.404,A 0.000,B 0.000,C 90.000,E1 288.725} C_DIS
LIN {X -0.344,Y -579.978,Z 522.397,A 0.000,B 0.000,C 90.000,E1 287.402} C_DIS
LIN {X 0.284,Y -579.845,Z 522.391,A 0.000,B 0.000,C 90.000,E1 286.260} C_DIS
LIN {X -0.152,Y -579.513,Z 522.383,A 0.000,B 0.000,C 90.000,E1 284.954} C_DIS
LIN {X -0.034,Y -579.170,Z 522.376,A 0.000,B 0.000,C 90.000,E1 283.592} C_DIS
LIN {X 0.164,Y -578.705,Z 522.367,A 0.000,B 0.000,C 90.000,E1 281.951} C_DIS
LIN {X -0.002,Y -578.040,Z 522.356,A 0.000,B 0.000,C 90.000,E1 280.074} C_DIS
LIN {X -0.253,Y -577.566,Z 522.349,A 0.000,B 0.000,C 90.000,E1 278.746} C_DIS
LIN {X -0.082,Y -576.922,Z 522.338,A 0.000,B 0.000,C 90.000,E1 276.834} C_DIS
LIN {X -0.209,Y -576.256,Z 522.329,A 0.000,B 0.000,C 90.000,E1 275.220} C_DIS
LIN {X 0.026,Y -575.531,Z 522.321,A 0.000,B 0.000,C 90.000,E1 273.841} C_DIS
LIN {X 0.213,Y -574.618,Z 522.314,A 0.000,B 0.000,C 90.000,E1 272.465} C_DIS
LIN {X -0.046,Y -573.364,Z 522.305,A 0.000,B 0.000,C 90.000,E1 270.859} C_DIS
LIN {X -0.049,Y -572.382,Z 522.299,A 0.000,B 0.000,C 90.000,E1 269.771} C_DIS
LIN {X 0.065,Y -571.127,Z 522.291,A 0.000,B 0.000,C 90.000,E1 268.396} C_DIS
LIN {X -0.242,Y -569.545,Z 522.282,A 0.000,B 0.000,C 90.000,E1 266.788} C_DIS
LIN {X -0.164,Y -568.194,Z 522.274,A 0.000,B 0.000,C 90.000,E1 265.412} C_DIS
LIN {X -0.076,Y -566.738,Z 522.267,A 0.000,B 0.000,C 90.000,E1 264.033} C_DIS
LIN {X -0.049,Y -565.480,Z 522.261,A 0.000,B 0.000,C 90.000,E1 262.932} C_DIS
LIN {X 0.055,Y -563.711,Z 522.253,A 0.000,B 0.000,C 90.000,E1 261.546} C_DIS
LIN {X -0.188,Y -561.533,Z 522.244,A 0.000,B 0.000,C 90.000,E1 259.916} C_DIS
LIN {X -0.075,Y -559.691,Z 522.236,A 0.000,B 0.000,C 90.000,E1 258.522} C_DIS
LIN {X -0.037,Y -558.114,Z 522.230,A 0.000,B 0.000,C 90.000,E1 257.409} C_DIS
LIN {X 0.239,Y -555.963,Z 522.222,A 0.000,B 0.000,C 90.000,E1 255.992} C_DIS
LIN {X -0.058,Y -553.636,Z 522.215,A 0.000,B 0.000,C 90.000,E1 254.629} C_DIS
LIN {X 0.019,Y -551.595,Z 522.208,A 0.000,B 0.000,C 90.000,E1 253.504} C_DIS
LIN {X -0.041,Y -549.931,Z 522.204,A 0.000,B 0.000,C 90.000,E1 252.670} C_DIS
LIN {X -0.133,Y -546.954,Z 522.196,A 0.000,B 0.000,C 90.000,E1 251.275} C_DIS
LIN {X 0.179,Y -544.489,Z 522.190,A 0.000,B 0.000,C 90.000,E1 250.115} C_DIS
LIN {X -0.245,Y -541.875,Z 522.183,A 0.000,B 0.000,C 90.000,E1 249.028} C_DIS
LIN {X 0.185,Y -539.133,Z 522.177,A 0.000,B 0.000,C 90.000,E1 247.847} C_DIS
LIN {X -0.127,Y -536.284,Z 522.171,A 0.000,B 0.000,C 90.000,E1 246.741} C_DIS
LIN {X 0.149,Y -532.493,Z 522.163,A 0.000,B 0.000,C 90.000,E1 245.281} C_DIS
LIN {X 0.130,Y -528.487,Z 522.155,A 0.000,B 0.000,C 90.000,E1 243.845} C_DIS
LIN {X 0.028,Y -524.363,Z 522.147,A 0.000,B 0.000,C 90.000,E1 242.410} C_DIS
LIN {X -0.134,Y -520.168,Z 522.139,A 0.000,B 0.000,C 90.000,E1 240.973} C_DIS
LIN {X 0.069,Y -515.913,Z 522.131,A 0.000,B 0.000,C 90.000,E1 239.488} C_DIS
LIN {X -0.084,Y -512.372,Z 522.124,A 0.000,B 0.000,C 90.000,E1 238.329} C_DIS
LIN {X -0.045,Y -506.820,Z 522.114,A 0.000,B 0.000,C 90.000,E1 236.548} C_DIS
LIN {X 0.039,Y -499.410,Z 522.101,A 0.000,B 0.000,C 90.000,E1 234.149} C_DIS
LIN {X -0.029,Y -492.535,Z 522.087,A 0.000,B 0.000,C 90.000,E1 231.743} C_DIS
LIN {X 0.043,Y -487.478,Z 522.077,A 0.000,B 0.000,C 90.000,E1 229.908} C_DIS
LIN {X -0.060,Y -482.513,Z 522.067,A 0.000,B 0.000,C 90.000,E1 228.081} C_DIS
LIN {X 0.134,Y -479.374,Z 522.060,A 0.000,B 0.000,C 90.000,E1 226.824} C_DIS
LIN {X -0.175,Y -474.633,Z 522.050,A 0.000,B 0.000,C 90.000,E1 225.000} C_DIS
LIN {X 0.223,Y -471.574,Z 522.043,A 0.000,B 0.000,C 90.000,E1 223.704} C_DIS
LIN {X 0.148,Y -466.265,Z 522.031,A 0.000,B 0.000,C 90.000,E1 221.515} C_DIS
LIN {X 0.130,Y -463.428,Z 522.024,A 0.000,B 0.000,C 90.000,E1 220.253} C_DIS
LIN {X -0.150,Y -459.155,Z 522.013,A 0.000,B 0.000,C 90.000,E1 218.382} C_DIS
LIN {X -0.185,Y -455.701,Z 522.004,A 0.000,B 0.000,C 90.000,E1 216.790} C_DIS
LIN {X -0.126,Y -450.986,Z 521.992,A 0.000,B 0.000,C 90.000,E1 214.532} C_DIS
LIN {X -0.013,Y -445.880,Z 521.977,A 0.000,B 0.000,C 90.000,E1 211.926} C_DIS
LIN {X -0.199,Y -441.572,Z 521.965,A 0.000,B 0.000,C 90.000,E1 209.667} C_DIS
LIN {X 0.196,Y -438.684,Z 521.956,A 0.000,B 0.000,C 90.000,E1 207.975} C_DIS
LIN {X -0.042,Y -435.245,Z 521.945,A 0.000,B 0.000,C 90.000,E1 206.027} C_DIS
LIN {X 0.046,Y -431.902,Z 521.934,A 0.000,B 0.000,C 90.000,E1 204.027} C_DIS
LIN {X 0.074,Y -427.660,Z 521.919,A 0.000,B 0.000,C 90.000,E1 201.354} C_DIS
LIN {X -0.131,Y -424.348,Z 521.906,A 0.000,B 0.000,C 90.000,E1 199.033} C_DIS
LIN {X 0.005,Y -420.834,Z 521.891,A 0.000,B 0.000,C 90.000,E1 196.315} C_DIS
LIN {X 0.213,Y -418.764,Z 521.881,A 0.000,B 0.000,C 90.000,E1 194.592} C_DIS
LIN {X 0.127,Y -417.108,Z 521.874,A 0.000,B 0.000,C 90.000,E1 193.244} C_DIS
LIN {X -0.154,Y -414.379,Z 521.860,A 0.000,B 0.000,C 90.000,E1 190.894} C_DIS
LIN {X 0.025,Y -412.948,Z 521.853,A 0.000,B 0.000,C 90.000,E1 189.500} C_DIS
LIN {X 0.214,Y -411.159,Z 521.843,A 0.000,B 0.000,C 90.000,E1 187.757} C_DIS
LIN {X -0.151,Y -409.332,Z 521.834,A 0.000,B 0.000,C 90.000,E1 186.087} C_DIS
LIN {X 0.147,Y -405.312,Z 521.809,A 0.000,B 0.000,C 90.000,E1 181.547} C_DIS
LIN {X -0.017,Y -403.930,Z 521.797,A 0.000,B 0.000,C 90.000,E1 179.484} C_DIS
LIN {X 0.063,Y -402.304,Z 521.778,A 0.000,B 0.000,C 90.000,E1 175.988} C_DIS
LIN {X -0.150,Y -401.653,Z 521.760,A 0.000,B 0.000,C 90.000,E1 172.875} C_DIS
LIN {X 0.134,Y -401.581,Z 521.745,A 0.000,B 0.000,C 90.000,E1 170.038} C_DIS
LIN {X -0.170,Y -401.976,Z 521.727,A 0.000,B 0.000,C 90.000,E1 166.937} C_DIS
LIN {X 0.140,Y -402.682,Z 521.714,A 0.000,B 0.000,C 90.000,E1 164.448} C_DIS
LIN {X -0.092,Y -403.880,Z 521.698,A 0.000,B 0.000,C 90.000,E1 161.692} C_DIS
LIN {X -0.038,Y -405.408,Z 521.683,A 0.000,B 0.000,C 90.000,E1 158.901} C_DIS
LIN {X 0.134,Y -406.756,Z 521.671,A 0.000,B 0.000,C 90.000,E1 156.794} C_DIS
LIN {X 0.130,Y -408.323,Z 521.660,A 0.000,B 0.000,C 90.000,E1 154.717} C_DIS
LIN {X 0.057,Y -409.667,Z 521.650,A 0.000,B 0.000,C 90.000,E1 152.999} C_DIS
LIN {X -0.093,Y -410.650,Z 521.642,A 0.000,B 0.000,C 90.000,E1 151.641} C_DIS
LIN {X -0.030,Y -411.645,Z 521.635,A 0.000,B 0.000,C 90.000,E1 150.255} C_DIS
LIN {X -0.018,Y -412.720,Z 521.625,A 0.000,B 0.000,C 90.000,E1 148.535} C_DIS
LIN {X -0.124,Y -413.667,Z 521.616,A 0.000,B 0.000,C 90.000,E1 146.834} C_DIS
LIN {X -0.047,Y -414.678,Z 521.604,A 0.000,B 0.000,C 90.000,E1 144.769} C_DIS
LIN {X -0.165,Y -415.283,Z 521.597,A 0.000,B 0.000,C 90.000,E1 143.417} C_DIS
LIN {X 0.128,Y -415.687,Z 521.591,A 0.000,B 0.000,C 90.000,E1 142.351} C_DIS
LIN {X 0.140,Y -416.272,Z 521.581,A 0.000,B 0.000,C 90.000,E1 140.642} C_DIS
LIN {X -0.019,Y -416.660,Z 521.574,A 0.000,B 0.000,C 90.000,E1 139.299} C_DIS
LIN {X 0.099,Y -416.955,Z 521.566,A 0.000,B 0.000,C 90.000,E1 137.919} C_DIS
LIN {X 0.096,Y -417.205,Z 521.557,A 0.000,B 0.000,C 90.000,E1 136.215} C_DIS
LIN {X 0.082,Y -417.197,Z 521.547,A 0.000,B 0.000,C 90.000,E1 134.514} C_DIS
LIN {X -0.100,Y -417.119,Z 521.540,A 0.000,B 0.000,C 90.000,E1 133.176} C_DIS
LIN {X 0.120,Y -416.910,Z 521.534,A 0.000,B 0.000,C 90.000,E1 132.123} C_DIS
LIN {X -0.224,Y -416.579,Z 521.529,A 0.000,B 0.000,C 90.000,E1 131.148} C_DIS
LIN {X 0.019,Y -416.043,Z 521.523,A 0.000,B 0.000,C 90.000,E1 130.092} C_DIS
LIN {X 0.032,Y -414.910,Z 521.513,A 0.000,B 0.000,C 90.000,E1 128.382} C_DIS
LIN {X -0.062,Y -413.700,Z 521.503,A 0.000,B 0.000,C 90.000,E1 126.583} C_DIS
LIN {X -0.101,Y -413.700,Z 521.503,A 0.000,B 0.000,C 90.000,E1 126.583} C_DIS
LIN {X -0.138,Y -415.472,Z 521.500,A 0.000,B 0.000,C 90.000,E1 126.011} C_DIS
LIN {X -0.079,Y -425.866,Z 521.477,A 0.000,B 0.000,C 90.000,E1 121.926} C_DIS
LIN {X -0.135,Y -430.888,Z 521.468,A 0.000,B 0.000,C 90.000,E1 120.256} C_DIS
LIN {X -0.206,Y -439.935,Z 521.448,A 0.000,B 0.000,C 90.000,E1 116.616} C_DIS
LIN {X -0.020,Y -444.728,Z 521.439,A 0.000,B 0.000,C 90.000,E1 114.951} C_DIS
LIN {X -0.108,Y -453.892,Z 521.417,A 0.000,B 0.000,C 90.000,E1 111.046} C_DIS
LIN {X -0.141,Y -453.972,Z 521.417,A 0.000,B 0.000,C 90.000,E1 111.046} C_DIS
LIN {X -0.058,Y -480.080,Z 521.412,A 0.000,B 0.000,C 90.000,E1 110.120} C_DIS
LIN {X -0.046,Y -494.081,Z 521.409,A 0.000,B 0.000,C 90.000,E1 109.631} C_DIS
LIN {X -0.196,Y -500.934,Z 521.408,A 0.000,B 0.000,C 90.000,E1 109.396} C_DIS
LIN {X -0.204,Y -518.233,Z 521.404,A 0.000,B 0.000,C 90.000,E1 108.725} C_DIS
LIN {X -0.038,Y -528.484,Z 521.402,A 0.000,B 0.000,C 90.000,E1 108.290} C_DIS
LIN {X 0.009,Y -535.181,Z 521.400,A 0.000,B 0.000,C 90.000,E1 108.000} C_DIS
LIN {X 0.133,Y -545.096,Z 521.398,A 0.000,B 0.000,C 90.000,E1 107.528} C_DIS
LIN {X -0.154,Y -551.374,Z 521.396,A 0.000,B 0.000,C 90.000,E1 107.221} C_DIS
LIN {X 0.161,Y -558.900,Z 521.393,A 0.000,B 0.000,C 90.000,E1 106.749} C_DIS
LIN {X -0.174,Y -563.341,Z 521.392,A 0.000,B 0.000,C 90.000,E1 106.496} C_DIS
LIN {X 0.167,Y -567.755,Z 521.390,A 0.000,B 0.000,C 90.000,E1 106.150} C_DIS
LIN {X -0.144,Y -572.104,Z 521.388,A 0.000,B 0.000,C 90.000,E1 105.843} C_DIS
LIN {X 0.055,Y -574.852,Z 521.387,A 0.000,B 0.000,C 90.000,E1 105.607} C_DIS
LIN {X 0.003,Y -579.696,Z 521.384,A 0.000,B 0.000,C 90.000,E1 105.190} C_DIS
LIN {X -0.117,Y -584.887,Z 521.382,A 0.000,B 0.000,C 90.000,E1 104.717} C_DIS
LIN {X 0.080,Y -589.809,Z 521.379,A 0.000,B 0.000,C 90.000,E1 104.189} C_DIS
LIN {X 0.051,Y -595.674,Z 521.375,A 0.000,B 0.000,C 90.000,E1 103.536} C_DIS
LIN {X -0.035,Y -601.125,Z 521.372,A 0.000,B 0.000,C 90.000,E1 102.883} C_DIS
LIN {X 0.313,Y -607.221,Z 521.367,A 0.000,B 0.000,C 90.000,E1 102.063} C_DIS
LIN {X 0.196,Y -612.076,Z 521.364,A 0.000,B 0.000,C 90.000,E1 101.422} C_DIS
LIN {X 0.241,Y -618.081,Z 521.359,A 0.000,B 0.000,C 90.000,E1 100.546} C_DIS
LIN {X 0.049,Y -622.898,Z 521.354,A 0.000,B 0.000,C 90.000,E1 99.792} C_DIS
LIN {X 0.065,Y -626.527,Z 521.351,A 0.000,B 0.000,C 90.000,E1 99.151} C_DIS
LIN {X -0.188,Y -629.352,Z 521.348,A 0.000,B 0.000,C 90.000,E1 98.681} C_DIS
LIN {X 0.254,Y -634.493,Z 521.343,A 0.000,B 0.000,C 90.000,E1 97.644} C_DIS
LIN {X -0.310,Y -637.634,Z 521.339,A 0.000,B 0.000,C 90.000,E1 97.068} C_DIS
LIN {X 0.063,Y -642.371,Z 521.334,A 0.000,B 0.000,C 90.000,E1 96.030} C_DIS
LIN {X 0.093,Y -645.687,Z 521.329,A 0.000,B 0.000,C 90.000,E1 95.277} C_DIS
LIN {X 0.092,Y -648.753,Z 521.325,A 0.000,B 0.000,C 90.000,E1 94.531} C_DIS
LIN {X 0.122,Y -651.526,Z 521.321,A 0.000,B 0.000,C 90.000,E1 93.784} C_DIS
LIN {X -0.092,Y -652.438,Z 521.320,A 0.000,B 0.000,C 90.000,E1 93.555} C_DIS
LIN {X -0.028,Y -654.699,Z 521.316,A 0.000,B 0.000,C 90.000,E1 92.808} C_DIS
LIN {X 0.226,Y -656.078,Z 521.313,A 0.000,B 0.000,C 90.000,E1 92.293} C_DIS
LIN {X -0.163,Y -657.204,Z 521.310,A 0.000,B 0.000,C 90.000,E1 91.835} C_DIS
LIN {X 0.131,Y -658.123,Z 521.307,A 0.000,B 0.000,C 90.000,E1 91.318} C_DIS
LIN {X 0.227,Y -659.097,Z 521.303,A 0.000,B 0.000,C 90.000,E1 90.573} C_DIS
LIN {X -0.140,Y -659.579,Z 521.301,A 0.000,B 0.000,C 90.000,E1 90.115} C_DIS
LIN {X -0.028,Y -659.798,Z 521.297,A 0.000,B 0.000,C 90.000,E1 89.370} C_DIS
LIN {X 0.086,Y -659.694,Z 521.292,A 0.000,B 0.000,C 90.000,E1 88.625} C_DIS
LIN {X -0.097,Y -659.601,Z 521.291,A 0.000,B 0.000,C 90.000,E1 88.396} C_DIS
LIN {X 0.033,Y -658.896,Z 521.287,A 0.000,B 0.000,C 90.000,E1 87.650} C_DIS
LIN {X 0.317,Y -658.265,Z 521.284,A 0.000,B 0.000,C 90.000,E1 87.135} C_DIS
LIN {X -0.216,Y -656.952,Z 521.280,A 0.000,B 0.000,C 90.000,E1 86.445} C_DIS
LIN {X 0.095,Y -655.959,Z 521.277,A 0.000,B 0.000,C 90.000,E1 85.927} C_DIS
LIN {X -0.302,Y -654.774,Z 521.275,A 0.000,B 0.000,C 90.000,E1 85.469} C_DIS
LIN {X -0.004,Y -653.457,Z 521.272,A 0.000,B 0.000,C 90.000,E1 84.951} C_DIS
LIN {X 0.287,Y -651.877,Z 521.269,A 0.000,B 0.000,C 90.000,E1 84.432} C_DIS
LIN {X -0.300,Y -649.333,Z 521.265,A 0.000,B 0.000,C 90.000,E1 83.742} C_DIS
LIN {X -0.037,Y -647.572,Z 521.262,A 0.000,B 0.000,C 90.000,E1 83.223} C_DIS
LIN {X 0.213,Y -645.582,Z 521.260,A 0.000,B 0.000,C 90.000,E1 82.704} C_DIS
LIN {X 0.283,Y -642.307,Z 521.255,A 0.000,B 0.000,C 90.000,E1 81.951} C_DIS
LIN {X 0.323,Y -638.811,Z 521.251,A 0.000,B 0.000,C 90.000,E1 81.197} C_DIS
LIN {X 0.181,Y -634.314,Z 521.246,A 0.000,B 0.000,C 90.000,E1 80.330} C_DIS
LIN {X 0.129,Y -630.043,Z 521.242,A 0.000,B 0.000,C 90.000,E1 79.577} C_DIS
LIN {X 0.312,Y -626.331,Z 521.239,A 0.000,B 0.000,C 90.000,E1 78.926} C_DIS
LIN {X 0.131,Y -620.585,Z 521.234,A 0.000,B 0.000,C 90.000,E1 78.049} C_DIS
LIN {X -0.262,Y -618.082,Z 521.232,A 0.000,B 0.000,C 90.000,E1 77.701} C_DIS
LIN {X 0.245,Y -612.446,Z 521.227,A 0.000,B 0.000,C 90.000,E1 76.881} C_DIS
LIN {X 0.292,Y -607.146,Z 521.224,A 0.000,B 0.000,C 90.000,E1 76.228} C_DIS
LIN {X -0.266,Y -601.293,Z 521.220,A 0.000,B 0.000,C 90.000,E1 75.644} C_DIS
LIN {X 0.133,Y -596.382,Z 521.217,A 0.000,B 0.000,C 90.000,E1 75.102} C_DIS
LIN {X 0.194,Y -591.485,Z 521.215,A 0.000,B 0.000,C 90.000,E1 74.629} C_DIS
LIN {X -0.017,Y -585.836,Z 521.212,A 0.000,B 0.000,C 90.000,E1 74.157} C_DIS
LIN {X 0.074,Y -579.933,Z 521.209,A 0.000,B 0.000,C 90.000,E1 73.685} C_DIS
LIN {X 0.255,Y -572.582,Z 521.207,A 0.000,B 0.000,C 90.000,E1 73.142} C_DIS
LIN {X 0.033,Y -567.698,Z 521.205,A 0.000,B 0.000,C 90.000,E1 72.851} C_DIS
LIN {X -0.237,Y -563.046,Z 521.203,A 0.000,B 0.000,C 90.000,E1 72.598} C_DIS
LIN {X 0.032,Y -558.208,Z 521.202,A 0.000,B 0.000,C 90.000,E1 72.308} C_DIS
LIN {X -0.168,Y -551.380,Z 521.200,A 0.000,B 0.000,C 90.000,E1 72.000} C_DIS
LIN {X -0.030,Y -544.020,Z 521.198,A 0.000,B 0.000,C 90.000,E1 71.692} C_DIS
LIN {X -0.270,Y -540.494,Z 521.198,A 0.000,B 0.000,C 90.000,E1 71.583} C_DIS
LIN {X -0.125,Y -533.267,Z 521.196,A 0.000,B 0.000,C 90.000,E1 71.329} C_DIS
LIN {X 0.047,Y -525.112,Z 521.195,A 0.000,B 0.000,C 90.000,E1 71.094} C_DIS
LIN {X 0.114,Y -512.620,Z 521.193,A 0.000,B 0.000,C 90.000,E1 70.786} C_DIS
LIN {X -0.138,Y -503.536,Z 521.192,A 0.000,B 0.000,C 90.000,E1 70.604} C_DIS
LIN {X 0.023,Y -491.289,Z 521.191,A 0.000,B 0.000,C 90.000,E1 70.369} C_DIS
LIN {X -0.093,Y -472.816,Z 521.189,A 0.000,B 0.000,C 90.000,E1 70.061} C_DIS
LIN {X 0.014,Y -470.223,Z 521.189,A 0.000,B 0.000,C 90.000,E1 70.007} C_DIS
LIN {X -0.019,Y -470.199,Z 521.189,A 0.000,B 0.000,C 90.000,E1 70.007} C_DIS
LIN {X -0.204,Y -465.774,Z 521.173,A 0.000,B 0.000,C 90.000,E1 67.177} C_DIS
LIN {X -0.141,Y -464.405,Z 521.170,A 0.000,B 0.000,C 90.000,E1 66.538} C_DIS
LIN {X 0.200,Y -456.260,Z 521.147,A 0.000,B 0.000,C 90.000,E1 62.359} C_DIS
LIN {X -0.206,Y -455.107,Z 521.143,A 0.000,B 0.000,C 90.000,E1 61.769} C_DIS
LIN {X -0.190,Y -446.009,Z 521.120,A 0.000,B 0.000,C 90.000,E1 57.661} C_DIS
LIN {X -0.230,Y -446.011,Z 521.120,A 0.000,B 0.000,C 90.000,E1 57.661} C_DIS
LIN {X -0.156,Y -448.233,Z 521.116,A 0.000,B 0.000,C 90.000,E1 56.914} C_DIS
LIN {X 0.016,Y -451.967,Z 521.109,A 0.000,B 0.000,C 90.000,E1 55.595} C_DIS
LIN {X 0.159,Y -454.460,Z 521.104,A 0.000,B 0.000,C 90.000,E1 54.609} C_DIS
LIN {X 0.061,Y -457.492,Z 521.096,A 0.000,B 0.000,C 90.000,E1 53.336} C_DIS
LIN {X -0.111,Y -458.881,Z 521.093,A 0.000,B 0.000,C 90.000,E1 52.718} C_DIS
LIN {X 0.024,Y -460.634,Z 521.088,A 0.000,B 0.000,C 90.000,E1 51.743} C_DIS
LIN {X -0.063,Y -462.676,Z 521.080,A 0.000,B 0.000,C 90.000,E1 50.481} C_DIS
LIN {X -0.171,Y -464.061,Z 521.075,A 0.000,B 0.000,C 90.000,E1 49.542} C_DIS
LIN {X 0.090,Y -465.647,Z 521.068,A 0.000,B 0.000,C 90.000,E1 48.243} C_DIS
LIN {X -0.036,Y -466.670,Z 521.063,A 0.000,B 0.000,C 90.000,E1 47.310} C_DIS
LIN {X -0.078,Y -467.738,Z 521.056,A 0.000,B 0.000,C 90.000,E1 46.053} C_DIS
LIN {X 0.220,Y -468.569,Z 521.049,A 0.000,B 0.000,C 90.000,E1 44.757} C_DIS
LIN {X -0.288,Y -468.894,Z 521.045,A 0.000,B 0.000,C 90.000,E1 44.190} C_DIS
LIN {X -0.055,Y -469.223,Z 521.040,A 0.000,B 0.000,C 90.000,E1 43.218} C_DIS
LIN {X -0.066,Y -469.443,Z 521.033,A 0.000,B 0.000,C 90.000,E1 41.962} C_DIS
LIN {X -0.035,Y -469.309,Z 521.026,A 0.000,B 0.000,C 90.000,E1 40.701} C_DIS
LIN {X 0.005,Y -469.018,Z 521.019,A 0.000,B 0.000,C 90.000,E1 39.439} C_DIS
LIN {X 0.040,Y -468.576,Z 521.012,A 0.000,B 0.000,C 90.000,E1 38.177} C_DIS
LIN {X -0.223,Y -468.079,Z 521.005,A 0.000,B 0.000,C 90.000,E1 36.950} C_DIS
LIN {X -0.081,Y -467.267,Z 520.996,A 0.000,B 0.000,C 90.000,E1 35.358} C_DIS
LIN {X 0.124,Y -466.589,Z 520.989,A 0.000,B 0.000,C 90.000,E1 34.072} C_DIS
LIN {X 0.088,Y -465.615,Z 520.981,A 0.000,B 0.000,C 90.000,E1 32.498} C_DIS
LIN {X 0.027,Y -464.644,Z 520.972,A 0.000,B 0.000,C 90.000,E1 30.924} C_DIS
LIN {X 0.097,Y -463.573,Z 520.963,A 0.000,B 0.000,C 90.000,E1 29.333} C_DIS
LIN {X 0.088,Y -461.841,Z 520.949,A 0.000,B 0.000,C 90.000,E1 26.796} C_DIS
LIN {X 0.021,Y -460.204,Z 520.935,A 0.000,B 0.000,C 90.000,E1 24.259} C_DIS
LIN {X -0.129,Y -459.507,Z 520.928,A 0.000,B 0.000,C 90.000,E1 23.003} C_DIS
LIN {X 0.043,Y -458.413,Z 520.914,A 0.000,B 0.000,C 90.000,E1 20.429} C_DIS
LIN {X -0.217,Y -457.680,Z 520.903,A 0.000,B 0.000,C 90.000,E1 18.544} C_DIS
LIN {X -0.097,Y -456.980,Z 520.889,A 0.000,B 0.000,C 90.000,E1 15.969} C_DIS
LIN {X -0.128,Y -456.713,Z 520.874,A 0.000,B 0.000,C 90.000,E1 13.411} C_DIS
LIN {X 0.183,Y -456.928,Z 520.862,A 0.000,B 0.000,C 90.000,E1 11.130} C_DIS
LIN {X 0.195,Y -457.457,Z 520.848,A 0.000,B 0.000,C 90.000,E1 8.568} C_DIS
LIN {X 0.027,Y -458.402,Z 520.834,A 0.000,B 0.000,C 90.000,E1 6.030} C_DIS
LIN {X -0.148,Y -459.853,Z 520.819,A 0.000,B 0.000,C 90.000,E1 3.498} C_DIS
LIN {X 0.167,Y -461.192,Z 520.809,A 0.000,B 0.000,C 90.000,E1 1.547} C_DIS
LIN {X -0.076,Y -463.023,Z 520.797,A 0.000,B 0.000,C 90.000,E1 359.484} C_DIS
LIN {X 0.058,Y -466.145,Z 520.781,A 0.000,B 0.000,C 90.000,E1 356.617} C_DIS
LIN {X -0.132,Y -468.874,Z 520.769,A 0.000,B 0.000,C 90.000,E1 354.432} C_DIS
LIN {X -0.067,Y -470.550,Z 520.762,A 0.000,B 0.000,C 90.000,E1 353.166} C_DIS
LIN {X 0.196,Y -473.158,Z 520.752,A 0.000,B 0.000,C 90.000,E1 351.254} C_DIS
LIN {X 0.053,Y -475.766,Z 520.741,A 0.000,B 0.000,C 90.000,E1 349.398} C_DIS
LIN {X -0.006,Y -479.104,Z 520.729,A 0.000,B 0.000,C 90.000,E1 347.229} C_DIS
LIN {X -0.155,Y -484.611,Z 520.712,A 0.000,B 0.000,C 90.000,E1 344.157} C_DIS
LIN {X -0.090,Y -488.314,Z 520.702,A 0.000,B 0.000,C 90.000,E1 342.308} C_DIS
LIN {X -0.134,Y -491.421,Z 520.693,A 0.000,B 0.000,C 90.000,E1 340.786} C_DIS
LIN {X -0.065,Y -495.135,Z 520.683,A 0.000,B 0.000,C 90.000,E1 338.954} C_DIS
LIN {X 0.207,Y -498.229,Z 520.675,A 0.000,B 0.000,C 90.000,E1 337.411} C_DIS
LIN {X 0.071,Y -501.209,Z 520.666,A 0.000,B 0.000,C 90.000,E1 335.921} C_DIS
LIN {X 0.190,Y -504.112,Z 520.658,A 0.000,B 0.000,C 90.000,E1 334.409} C_DIS
LIN {X 0.215,Y -507.547,Z 520.648,A 0.000,B 0.000,C 90.000,E1 332.615} C_DIS
LIN {X -0.229,Y -510.369,Z 520.640,A 0.000,B 0.000,C 90.000,E1 331.179} C_DIS
LIN {X -0.020,Y -514.961,Z 520.627,A 0.000,B 0.000,C 90.000,E1 328.791} C_DIS
LIN {X -0.149,Y -518.473,Z 520.617,A 0.000,B 0.000,C 90.000,E1 327.041} C_DIS
LIN {X -0.250,Y -520.805,Z 520.610,A 0.000,B 0.000,C 90.000,E1 325.881} C_DIS
LIN {X -0.069,Y -523.730,Z 520.602,A 0.000,B 0.000,C 90.000,E1 324.402} C_DIS
LIN {X 0.107,Y -527.831,Z 520.591,A 0.000,B 0.000,C 90.000,E1 322.351} C_DIS
LIN {X -0.095,Y -530.783,Z 520.583,A 0.000,B 0.000,C 90.000,E1 320.928} C_DIS
LIN {X 0.161,Y -534.248,Z 520.573,A 0.000,B 0.000,C 90.000,E1 319.175} C_DIS
LIN {X 0.030,Y -537.240,Z 520.565,A 0.000,B 0.000,C 90.000,E1 317.757} C_DIS
LIN {X -0.014,Y -539.658,Z 520.559,A 0.000,B 0.000,C 90.000,E1 316.620} C_DIS
LIN {X -0.045,Y -544.265,Z 520.546,A 0.000,B 0.000,C 90.000,E1 314.352} C_DIS
LIN {X 0.040,Y -548.179,Z 520.535,A 0.000,B 0.000,C 90.000,E1 312.366} C_DIS
LIN {X 0.316,Y -553.161,Z 520.523,A 0.000,B 0.000,C 90.000,E1 310.092} C_DIS
LIN {X -0.129,Y -556.859,Z 520.514,A 0.000,B 0.000,C 90.000,E1 308.463} C_DIS
LIN {X -0.243,Y -559.054,Z 520.508,A 0.000,B 0.000,C 90.000,E1 307.363} C_DIS
LIN {X 0.174,Y -565.281,Z 520.491,A 0.000,B 0.000,C 90.000,E1 304.278} C_DIS
LIN {X -0.079,Y -566.666,Z 520.488,A 0.000,B 0.000,C 90.000,E1 303.754} C_DIS
LIN {X -0.283,Y -567.316,Z 520.486,A 0.000,B 0.000,C 90.000,E1 303.499} C_DIS
LIN {X 0.110,Y -568.876,Z 520.483,A 0.000,B 0.000,C 90.000,E1 302.911} C_DIS
LIN {X 0.346,Y -570.336,Z 520.480,A 0.000,B 0.000,C 90.000,E1 302.339} C_DIS
LIN {X 0.163,Y -571.202,Z 520.478,A 0.000,B 0.000,C 90.000,E1 302.084} C_DIS
LIN {X 0.265,Y -574.502,Z 520.474,A 0.000,B 0.000,C 90.000,E1 301.258} C_DIS
LIN {X -0.034,Y -579.847,Z 520.468,A 0.000,B 0.000,C 90.000,E1 300.207} C_DIS
LIN {X 0.172,Y -581.687,Z 520.466,A 0.000,B 0.000,C 90.000,E1 299.922} C_DIS
LIN {X 0.032,Y -582.744,Z 520.465,A 0.000,B 0.000,C 90.000,E1 299.667} C_DIS
LIN {X 0.137,Y -591.484,Z 520.456,A 0.000,B 0.000,C 90.000,E1 298.052} C_DIS
LIN {X 0.212,Y -594.151,Z 520.453,A 0.000,B 0.000,C 90.000,E1 297.513} C_DIS
LIN {X 0.118,Y -595.373,Z 520.452,A 0.000,B 0.000,C 90.000,E1 297.257} C_DIS
LIN {X -0.146,Y -597.723,Z 520.447,A 0.000,B 0.000,C 90.000,E1 296.488} C_DIS
LIN {X -0.229,Y -598.216,Z 520.446,A 0.000,B 0.000,C 90.000,E1 296.232} C_DIS
LIN {X 0.152,Y -598.838,Z 520.443,A 0.000,B 0.000,C 90.000,E1 295.668} C_DIS
LIN {X -0.001,Y -598.571,Z 520.440,A 0.000,B 0.000,C 90.000,E1 295.155} C_DIS
LIN {X -0.079,Y -598.143,Z 520.438,A 0.000,B 0.000,C 90.000,E1 294.899} C_DIS
LIN {X -0.237,Y -596.127,Z 520.435,A 0.000,B 0.000,C 90.000,E1 294.387} C_DIS
LIN {X 0.263,Y -595.436,Z 520.435,A 0.000,B 0.000,C 90.000,E1 294.207} C_DIS
LIN {X 0.221,Y -594.528,Z 520.434,A 0.000,B 0.000,C 90.000,E1 294.079} C_DIS
LIN {X 0.080,Y -590.987,Z 520.432,A 0.000,B 0.000,C 90.000,E1 293.695} C_DIS
LIN {X -0.018,Y -587.740,Z 520.430,A 0.000,B 0.000,C 90.000,E1 293.462} C_DIS
LIN {X 0.181,Y -585.532,Z 520.429,A 0.000,B 0.000,C 90.000,E1 293.206} C_DIS
LIN {X 0.120,Y -583.925,Z 520.428,A 0.000,B 0.000,C 90.000,E1 293.078} C_DIS
LIN {X -0.006,Y -581.815,Z 520.427,A 0.000,B 0.000,C 90.000,E1 292.823} C_DIS
LIN {X -0.072,Y -581.046,Z 520.426,A 0.000,B 0.000,C 90.000,E1 292.695} C_DIS
LIN {X -0.326,Y -580.603,Z 520.425,A 0.000,B 0.000,C 90.000,E1 292.589} C_DIS
LIN {X 0.070,Y -580.262,Z 520.424,A 0.000,B 0.000,C 90.000,E1 292.280} C_DIS
LIN {X -0.221,Y -580.026,Z 520.421,A 0.000,B 0.000,C 90.000,E1 291.770} C_DIS
LIN {X -0.067,Y -580.770,Z 520.410,A 0.000,B 0.000,C 90.000,E1 289.866} C_DIS
LIN {X 0.016,Y -581.013,Z 520.404,A 0.000,B 0.000,C 90.000,E1 288.779} C_DIS
LIN {X -0.238,Y -581.112,Z 520.397,A 0.000,B 0.000,C 90.000,E1 287.457} C_DIS
LIN {X 0.063,Y -580.946,Z 520.389,A 0.000,B 0.000,C 90.000,E1 286.079} C_DIS
LIN {X -0.133,Y -580.586,Z 520.380,A 0.000,B 0.000,C 90.000,E1 284.481} C_DIS
LIN {X -0.222,Y -580.321,Z 520.374,A 0.000,B 0.000,C 90.000,E1 283.411} C_DIS
LIN {X 0.113,Y -580.071,Z 520.368,A 0.000,B 0.000,C 90.000,E1 282.299} C_DIS
LIN {X -0.021,Y -579.466,Z 520.358,A 0.000,B 0.000,C 90.000,E1 280.423} C_DIS
LIN {X -0.030,Y -578.938,Z 520.349,A 0.000,B 0.000,C 90.000,E1 278.803} C_DIS
LIN {X 0.172,Y -578.314,Z 520.338,A 0.000,B 0.000,C 90.000,E1 276.891} C_DIS
LIN {X -0.130,Y -577.770,Z 520.331,A 0.000,B 0.000,C 90.000,E1 275.568} C_DIS
LIN {X 0.140,Y -577.063,Z 520.323,A 0.000,B 0.000,C 90.000,E1 274.188} C_DIS
LIN {X 0.240,Y -576.366,Z 520.317,A 0.000,B 0.000,C 90.000,E1 273.094} C_DIS
LIN {X 0.268,Y -575.564,Z 520.311,A 0.000,B 0.000,C 90.000,E1 272.007} C_DIS
LIN {X 0.029,Y -574.260,Z 520.302,A 0.000,B 0.000,C 90.000,E1 270.401} C_DIS
LIN {X -0.251,Y -572.661,Z 520.293,A 0.000,B 0.000,C 90.000,E1 268.797} C_DIS
LIN {X -0.251,Y -571.574,Z 520.287,A 0.000,B 0.000,C 90.000,E1 267.707} C_DIS
LIN {X 0.157,Y -569.693,Z 520.277,A 0.000,B 0.000,C 90.000,E1 265.755} C_DIS
LIN {X -0.177,Y -567.895,Z 520.267,A 0.000,B 0.000,C 90.000,E1 264.147} C_DIS
LIN {X -0.034,Y -566.256,Z 520.260,A 0.000,B 0.000,C 90.000,E1 262.761} C_DIS
LIN {X 0.078,Y -564.408,Z 520.252,A 0.000,B 0.000,C 90.000,E1 261.376} C_DIS
LIN {X 0.237,Y -562.539,Z 520.245,A 0.000,B 0.000,C 90.000,E1 259.982} C_DIS
LIN {X -0.084,Y -560.681,Z 520.237,A 0.000,B 0.000,C 90.000,E1 258.634} C_DIS
LIN {X -0.027,Y -559.058,Z 520.231,A 0.000,B 0.000,C 90.000,E1 257.521} C_DIS
LIN {X 0.140,Y -556.880,Z 520.223,A 0.000,B 0.000,C 90.000,E1 256.117} C_DIS
LIN {X 0.263,Y -555.001,Z 520.217,A 0.000,B 0.000,C 90.000,E1 254.991} C_DIS
LIN {X -0.174,Y -553.014,Z 520.211,A 0.000,B 0.000,C 90.000,E1 253.921} C_DIS
LIN {X 0.048,Y -550.805,Z 520.204,A 0.000,B 0.000,C 90.000,E1 252.779} C_DIS
LIN {X 0.239,Y -548.419,Z 520.198,A 0.000,B 0.000,C 90.000,E1 251.638} C_DIS
LIN {X -0.126,Y -545.948,Z 520.192,A 0.000,B 0.000,C 90.000,E1 250.550} C_DIS
LIN {X 0.169,Y -543.352,Z 520.186,A 0.000,B 0.000,C 90.000,E1 249.390} C_DIS
LIN {X -0.082,Y -540.613,Z 520.179,A 0.000,B 0.000,C 90.000,E1 248.284} C_DIS
LIN {X 0.332,Y -537.773,Z 520.173,A 0.000,B 0.000,C 90.000,E1 247.102} C_DIS
LIN {X -0.069,Y -533.988,Z 520.165,A 0.000,B 0.000,C 90.000,E1 245.717} C_DIS
LIN {X 0.240,Y -530.829,Z 520.159,A 0.000,B 0.000,C 90.000,E1 244.537} C_DIS
LIN {X 0.242,Y -527.582,Z 520.152,A 0.000,B 0.000,C 90.000,E1 243.384} C_DIS
LIN {X 0.278,Y -522.560,Z 520.143,A 0.000,B 0.000,C 90.000,E1 241.641} C_DIS
LIN {X 0.000,Y -517.447,Z 520.133,A 0.000,B 0.000,C 90.000,E1 239.921} C_DIS
LIN {X 0.050,Y -513.925,Z 520.126,A 0.000,B 0.000,C 90.000,E1 238.742} C_DIS
LIN {X -0.127,Y -510.234,Z 520.120,A 0.000,B 0.000,C 90.000,E1 237.582} C_DIS
LIN {X 0.070,Y -506.514,Z 520.113,A 0.000,B 0.000,C 90.000,E1 236.373} C_DIS
LIN {X 0.132,Y -499.979,Z 520.102,A 0.000,B 0.000,C 90.000,E1 234.276} C_DIS
LIN {X -0.056,Y -492.184,Z 520.087,A 0.000,B 0.000,C 90.000,E1 231.582} C_DIS
LIN {X 0.012,Y -487.163,Z 520.076,A 0.000,B 0.000,C 90.000,E1 229.747} C_DIS
LIN {X 0.039,Y -481.418,Z 520.065,A 0.000,B 0.000,C 90.000,E1 227.595} C_DIS
LIN {X 0.097,Y -479.037,Z 520.059,A 0.000,B 0.000,C 90.000,E1 226.662} C_DIS
LIN {X 0.010,Y -475.110,Z 520.051,A 0.000,B 0.000,C 90.000,E1 225.121} C_DIS
LIN {X -0.059,Y -470.441,Z 520.040,A 0.000,B 0.000,C 90.000,E1 223.257} C_DIS
LIN {X 0.022,Y -466.699,Z 520.032,A 0.000,B 0.000,C 90.000,E1 221.676} C_DIS
LIN {X 0.065,Y -463.102,Z 520.023,A 0.000,B 0.000,C 90.000,E1 220.092} C_DIS
LIN {X -0.254,Y -459.566,Z 520.014,A 0.000,B 0.000,C 90.000,E1 218.543} C_DIS
LIN {X 0.095,Y -455.428,Z 520.003,A 0.000,B 0.000,C 90.000,E1 216.583} C_DIS
LIN {X -0.195,Y -451.397,Z 519.993,A 0.000,B 0.000,C 90.000,E1 214.692} C_DIS
LIN {X -0.057,Y -446.270,Z 519.978,A 0.000,B 0.000,C 90.000,E1 212.084} C_DIS
LIN {X -0.055,Y -442.593,Z 519.967,A 0.000,B 0.000,C 90.000,E1 210.129} C_DIS
LIN {X 0.012,Y -439.062,Z 519.956,A 0.000,B 0.000,C 90.000,E1 208.153} C_DIS
LIN {X -0.023,Y -435.611,Z 519.945,A 0.000,B 0.000,C 90.000,E1 206.181} C_DIS
LIN {X -0.130,Y -432.268,Z 519.934,A 0.000,B 0.000,C 90.000,E1 204.207} C_DIS
LIN {X 0.098,Y -428.485,Z 519.922,A 0.000,B 0.000,C 90.000,E1 201.844} C_DIS
LIN {X 0.056,Y -425.100,Z 519.908,A 0.000,B 0.000,C 90.000,E1 199.504} C_DIS
LIN {X 0.083,Y -421.499,Z 519.893,A 0.000,B 0.000,C 90.000,E1 196.804} C_DIS
LIN {X -0.093,Y -419.421,Z 519.884,A 0.000,B 0.000,C 90.000,E1 195.134} C_DIS
LIN {X 0.142,Y -416.955,Z 519.873,A 0.000,B 0.000,C 90.000,E1 193.063} C_DIS
LIN {X -0.150,Y -414.266,Z 519.859,A 0.000,B 0.000,C 90.000,E1 190.715} C_DIS
LIN {X 0.062,Y -412.449,Z 519.850,A 0.000,B 0.000,C 90.000,E1 188.973} C_DIS
LIN {X 0.178,Y -410.733,Z 519.840,A 0.000,B 0.000,C 90.000,E1 187.239} C_DIS
LIN {X -0.174,Y -408.466,Z 519.829,A 0.000,B 0.000,C 90.000,E1 185.220} C_DIS
LIN {X 0.085,Y -405.262,Z 519.808,A 0.000,B 0.000,C 90.000,E1 181.375} C_DIS
LIN {X -0.080,Y -403.894,Z 519.796,A 0.000,B 0.000,C 90.000,E1 179.312} C_DIS
LIN {X -0.019,Y -402.240,Z 519.775,A 0.000,B 0.000,C 90.000,E1 175.469} C_DIS
LIN {X 0.169,Y -401.674,Z 519.757,A 0.000,B 0.000,C 90.000,E1 172.299} C_DIS
LIN {X 0.127,Y -401.697,Z 519.744,A 0.000,B 0.000,C 90.000,E1 169.859} C_DIS
LIN {X -0.175,Y -402.217,Z 519.724,A 0.000,B 0.000,C 90.000,E1 166.408} C_DIS
LIN {X 0.046,Y -402.865,Z 519.713,A 0.000,B 0.000,C 90.000,E1 164.283} C_DIS
LIN {X 0.213,Y -403.928,Z 519.699,A 0.000,B 0.000,C 90.000,E1 161.819} C_DIS
LIN {X -0.114,Y -405.461,Z 519.684,A 0.000,B 0.000,C 90.000,E1 159.082} C_DIS
LIN {X -0.106,Y -407.343,Z 519.668,A 0.000,B 0.000,C 90.000,E1 156.305} C_DIS
LIN {X 0.082,Y -409.499,Z 519.653,A 0.000,B 0.000,C 90.000,E1 153.512} C_DIS
LIN {X -0.069,Y -410.534,Z 519.645,A 0.000,B 0.000,C 90.000,E1 152.153} C_DIS
LIN {X 0.079,Y -411.799,Z 519.636,A 0.000,B 0.000,C 90.000,E1 150.411} C_DIS
LIN {X 0.235,Y -413.099,Z 519.624,A 0.000,B 0.000,C 90.000,E1 148.329} C_DIS
LIN {X -0.024,Y -413.874,Z 519.617,A 0.000,B 0.000,C 90.000,E1 146.993} C_DIS
LIN {X 0.051,Y -414.934,Z 519.605,A 0.000,B 0.000,C 90.000,E1 144.928} C_DIS
LIN {X 0.114,Y -415.764,Z 519.596,A 0.000,B 0.000,C 90.000,E1 143.210} C_DIS
LIN {X 0.009,Y -416.316,Z 519.588,A 0.000,B 0.000,C 90.000,E1 141.859} C_DIS
LIN {X 0.030,Y -416.889,Z 519.579,A 0.000,B 0.000,C 90.000,E1 140.150} C_DIS
LIN {X 0.022,Y -417.387,Z 519.569,A 0.000,B 0.000,C 90.000,E1 138.447} C_DIS
LIN {X 0.152,Y -417.635,Z 519.562,A 0.000,B 0.000,C 90.000,E1 137.067} C_DIS
LIN {X -0.022,Y -417.766,Z 519.554,A 0.000,B 0.000,C 90.000,E1 135.729} C_DIS
LIN {X 0.095,Y -417.762,Z 519.547,A 0.000,B 0.000,C 90.000,E1 134.352} C_DIS
LIN {X 0.040,Y -417.706,Z 519.541,A 0.000,B 0.000,C 90.000,E1 133.338} C_DIS
LIN {X -0.133,Y -417.409,Z 519.533,A 0.000,B 0.000,C 90.000,E1 132.000} C_DIS
LIN {X -0.193,Y -416.999,Z 519.528,A 0.000,B 0.000,C 90.000,E1 130.987} C_DIS
LIN {X 0.052,Y -416.410,Z 519.522,A 0.000,B 0.000,C 90.000,E1 129.930} C_DIS
LIN {X 0.069,Y -415.237,Z 519.512,A 0.000,B 0.000,C 90.000,E1 128.222} C_DIS
LIN {X 0.078,Y -414.015,Z 519.503,A 0.000,B 0.000,C 90.000,E1 126.457} C_DIS
LIN {X 0.040,Y -414.023,Z 519.503,A 0.000,B 0.000,C 90.000,E1 126.457} C_DIS
LIN {X 0.239,Y -415.866,Z 519.499,A 0.000,B 0.000,C 90.000,E1 125.804} C_DIS
LIN {X 0.122,Y -425.338,Z 519.478,A 0.000,B 0.000,C 90.000,E1 122.084} C_DIS
LIN {X 0.066,Y -430.350,Z 519.469,A 0.000,B 0.000,C 90.000,E1 120.413} C_DIS
LIN {X 0.070,Y -431.968,Z 519.465,A 0.000,B 0.000,C 90.000,E1 119.745} C_DIS
LIN {X 0.064,Y -441.283,Z 519.445,A 0.000,B 0.000,C 90.000,E1 116.104} C_DIS
LIN {X -0.211,Y -444.184,Z 519.440,A 0.000,B 0.000,C 90.000,E1 115.155} C_DIS
LIN {X 0.233,Y -445.066,Z 519.438,A 0.000,B 0.000,C 90.000,E1 114.771} C_DIS
LIN {X -0.083,Y -454.223,Z 519.416,A 0.000,B 0.000,C 90.000,E1 110.918} C_DIS
LIN {X -0.283,Y -454.778,Z 519.415,A 0.000,B 0.000,C 90.000,E1 110.737} C_DIS
LIN {X 0.103,Y -454.883,Z 519.415,A 0.000,B 0.000,C 90.000,E1 110.684} C_DIS
LIN {X -0.032,Y -479.432,Z 519.410,A 0.000,B 0.000,C 90.000,E1 109.866} C_DIS
LIN {X 0.024,Y -489.989,Z 519.408,A 0.000,B 0.000,C 90.000,E1 109.504} C_DIS
LIN {X -0.050,Y -500.321,Z 519.406,A 0.000,B 0.000,C 90.000,E1 109.141} C_DIS
LIN {X -0.095,Y -517.656,Z 519.403,A 0.000,B 0.000,C 90.000,E1 108.489} C_DIS
LIN {X 0.163,Y -527.951,Z 519.400,A 0.000,B 0.000,C 90.000,E1 108.055} C_DIS
LIN {X -0.229,Y -534.626,Z 519.399,A 0.000,B 0.000,C 90.000,E1 107.819} C_DIS
LIN {X 0.134,Y -544.500,Z 519.396,A 0.000,B 0.000,C 90.000,E1 107.330} C_DIS
LIN {X -0.169,Y -550.689,Z 519.395,A 0.000,B 0.000,C 90.000,E1 107.040} C_DIS
LIN {X 0.019,Y -559.958,Z 519.392,A 0.000,B 0.000,C 90.000,E1 106.496} C_DIS
LIN {X -0.169,Y -567.272,Z 519.389,A 0.000,B 0.000,C 90.000,E1 106.024} C_DIS
LIN {X 0.177,Y -573.173,Z 519.387,A 0.000,B 0.000,C 90.000,E1 105.552} C_DIS
LIN {X -0.058,Y -578.555,Z 519.384,A 0.000,B 0.000,C 90.000,E1 105.134} C_DIS
LIN {X -0.022,Y -583.925,Z 519.381,A 0.000,B 0.000,C 90.000,E1 104.647} C_DIS
LIN {X -0.022,Y -590.219,Z 519.378,A 0.000,B 0.000,C 90.000,E1 104.008} C_DIS
LIN {X -0.037,Y -595.079,Z 519.375,A 0.000,B 0.000,C 90.000,E1 103.480} C_DIS
LIN {X 0.105,Y -602.439,Z 519.370,A 0.000,B 0.000,C 90.000,E1 102.591} C_DIS
LIN {X -0.322,Y -609.654,Z 519.365,A 0.000,B 0.000,C 90.000,E1 101.715} C_DIS
LIN {X -0.291,Y -615.963,Z 519.360,A 0.000,B 0.000,C 90.000,E1 100.838} C_DIS
LIN {X -0.166,Y -619.484,Z 519.357,A 0.000,B 0.000,C 90.000,E1 100.310} C_DIS
LIN {X 0.268,Y -624.369,Z 519.353,A 0.000,B 0.000,C 90.000,E1 99.500} C_DIS
LIN {X 0.267,Y -629.437,Z 519.348,A 0.000,B 0.000,C 90.000,E1 98.624} C_DIS
LIN {X 0.185,Y -633.509,Z 519.344,A 0.000,B 0.000,C 90.000,E1 97.871} C_DIS
LIN {X -0.132,Y -638.688,Z 519.338,A 0.000,B 0.000,C 90.000,E1 96.891} C_DIS
LIN {X -0.201,Y -642.273,Z 519.334,A 0.000,B 0.000,C 90.000,E1 96.144} C_DIS
LIN {X 0.231,Y -646.702,Z 519.329,A 0.000,B 0.000,C 90.000,E1 95.106} C_DIS
LIN {X -0.179,Y -648.793,Z 519.326,A 0.000,B 0.000,C 90.000,E1 94.645} C_DIS
LIN {X 0.285,Y -652.525,Z 519.320,A 0.000,B 0.000,C 90.000,E1 93.612} C_DIS
LIN {X -0.301,Y -654.885,Z 519.316,A 0.000,B 0.000,C 90.000,E1 92.922} C_DIS
LIN {X -0.048,Y -656.300,Z 519.313,A 0.000,B 0.000,C 90.000,E1 92.407} C_DIS
LIN {X 0.049,Y -657.949,Z 519.309,A 0.000,B 0.000,C 90.000,E1 91.661} C_DIS
LIN {X 0.329,Y -658.838,Z 519.307,A 0.000,B 0.000,C 90.000,E1 91.146} C_DIS
LIN {X -0.043,Y -659.468,Z 519.304,A 0.000,B 0.000,C 90.000,E1 90.688} C_DIS
LIN {X 0.251,Y -659.948,Z 519.301,A 0.000,B 0.000,C 90.000,E1 90.172} C_DIS
LIN {X -0.292,Y -660.224,Z 519.297,A 0.000,B 0.000,C 90.000,E1 89.484} C_DIS
LIN {X -0.175,Y -660.119,Z 519.293,A 0.000,B 0.000,C 90.000,E1 88.740} C_DIS
LIN {X 0.303,Y -660.054,Z 519.292,A 0.000,B 0.000,C 90.000,E1 88.453} C_DIS
LIN {X -0.221,Y -659.375,Z 519.288,A 0.000,B 0.000,C 90.000,E1 87.764} C_DIS
LIN {X 0.068,Y -658.786,Z 519.285,A 0.000,B 0.000,C 90.000,E1 87.249} C_DIS
LIN {X 0.196,Y -657.445,Z 519.281,A 0.000,B 0.000,C 90.000,E1 86.502} C_DIS
LIN {X 0.315,Y -655.894,Z 519.277,A 0.000,B 0.000,C 90.000,E1 85.755} C_DIS
LIN {X -0.085,Y -654.617,Z 519.274,A 0.000,B 0.000,C 90.000,E1 85.298} C_DIS
LIN {X -0.234,Y -653.940,Z 519.273,A 0.000,B 0.000,C 90.000,E1 85.065} C_DIS
LIN {X 0.279,Y -650.579,Z 519.267,A 0.000,B 0.000,C 90.000,E1 84.033} C_DIS
LIN {X -0.251,Y -647.904,Z 519.263,A 0.000,B 0.000,C 90.000,E1 83.337} C_DIS
LIN {X -0.237,Y -644.748,Z 519.259,A 0.000,B 0.000,C 90.000,E1 82.591} C_DIS
LIN {X -0.048,Y -641.895,Z 519.255,A 0.000,B 0.000,C 90.000,E1 81.951} C_DIS
LIN {X -0.012,Y -638.284,Z 519.251,A 0.000,B 0.000,C 90.000,E1 81.197} C_DIS
LIN {X -0.016,Y -634.275,Z 519.247,A 0.000,B 0.000,C 90.000,E1 80.443} C_DIS
LIN {X 0.088,Y -630.666,Z 519.243,A 0.000,B 0.000,C 90.000,E1 79.803} C_DIS
LIN {X 0.002,Y -626.052,Z 519.239,A 0.000,B 0.000,C 90.000,E1 79.050} C_DIS
LIN {X -0.068,Y -623.014,Z 519.237,A 0.000,B 0.000,C 90.000,E1 78.578} C_DIS
LIN {X 0.029,Y -617.973,Z 519.232,A 0.000,B 0.000,C 90.000,E1 77.813} C_DIS
LIN {X 0.005,Y -612.424,Z 519.228,A 0.000,B 0.000,C 90.000,E1 77.061} C_DIS
LIN {X 0.051,Y -607.077,Z 519.225,A 0.000,B 0.000,C 90.000,E1 76.408} C_DIS
LIN {X 0.079,Y -600.959,Z 519.221,A 0.000,B 0.000,C 90.000,E1 75.755} C_DIS
LIN {X 0.212,Y -595.877,Z 519.218,A 0.000,B 0.000,C 90.000,E1 75.227} C_DIS
LIN {X -0.019,Y -590.485,Z 519.215,A 0.000,B 0.000,C 90.000,E1 74.755} C_DIS
LIN {X -0.082,Y -584.865,Z 519.213,A 0.000,B 0.000,C 90.000,E1 74.283} C_DIS
LIN {X 0.120,Y -580.474,Z 519.211,A 0.000,B 0.000,C 90.000,E1 73.921} C_DIS
LIN {X -0.023,Y -574.442,Z 519.208,A 0.000,B 0.000,C 90.000,E1 73.504} C_DIS
LIN {X 0.055,Y -568.084,Z 519.206,A 0.000,B 0.000,C 90.000,E1 73.087} C_DIS
LIN {X 0.215,Y -563.082,Z 519.205,A 0.000,B 0.000,C 90.000,E1 72.779} C_DIS
LIN {X -0.129,Y -558.016,Z 519.203,A 0.000,B 0.000,C 90.000,E1 72.543} C_DIS
LIN {X 0.183,Y -551.092,Z 519.201,A 0.000,B 0.000,C 90.000,E1 72.181} C_DIS
LIN {X -0.212,Y -543.928,Z 519.200,A 0.000,B 0.000,C 90.000,E1 71.945} C_DIS
LIN {X -0.292,Y -538.608,Z 519.199,A 0.000,B 0.000,C 90.000,E1 71.764} C_DIS
LIN {X -0.270,Y -532.890,Z 519.198,A 0.000,B 0.000,C 90.000,E1 71.583} C_DIS
LIN {X 0.053,Y -525.321,Z 519.196,A 0.000,B 0.000,C 90.000,E1 71.348} C_DIS
LIN {X 0.088,Y -517.611,Z 519.195,A 0.000,B 0.000,C 90.000,E1 71.167} C_DIS
LIN {X 0.023,Y -502.924,Z 519.194,A 0.000,B 0.000,C 90.000,E1 70.859} C_DIS
LIN {X 0.177,Y -485.732,Z 519.192,A 0.000,B 0.000,C 90.000,E1 70.550} C_DIS
LIN {X -0.228,Y -471.026,Z 519.191,A 0.000,B 0.000,C 90.000,E1 70.369} C_DIS
LIN {X -0.259,Y -470.799,Z 519.191,A 0.000,B 0.000,C 90.000,E1 70.369} C_DIS
LIN {X 0.083,Y -465.642,Z 519.173,A 0.000,B 0.000,C 90.000,E1 67.050} C_DIS
LIN {X -0.039,Y -456.636,Z 519.148,A 0.000,B 0.000,C 90.000,E1 62.615} C_DIS
LIN {X -0.039,Y -455.592,Z 519.144,A 0.000,B 0.000,C 90.000,E1 61.975} C_DIS
LIN {X 0.145,Y -452.502,Z 519.137,A 0.000,B 0.000,C 90.000,E1 60.667} C_DIS
LIN {X 0.251,Y -446.360,Z 519.121,A 0.000,B 0.000,C 90.000,E1 57.788} C_DIS
LIN {X 0.211,Y -446.354,Z 519.121,A 0.000,B 0.000,C 90.000,E1 57.788} C_DIS
LIN {X 0.028,Y -448.569,Z 519.117,A 0.000,B 0.000,C 90.000,E1 57.120} C_DIS
LIN {X 0.206,Y -452.398,Z 519.110,A 0.000,B 0.000,C 90.000,E1 55.801} C_DIS
LIN {X 0.094,Y -455.034,Z 519.105,A 0.000,B 0.000,C 90.000,E1 54.848} C_DIS
LIN {X -0.002,Y -458.122,Z 519.098,A 0.000,B 0.000,C 90.000,E1 53.577} C_DIS
LIN {X -0.159,Y -460.183,Z 519.092,A 0.000,B 0.000,C 90.000,E1 52.637} C_DIS
LIN {X -0.034,Y -461.391,Z 519.089,A 0.000,B 0.000,C 90.000,E1 51.984} C_DIS
LIN {X -0.116,Y -463.423,Z 519.082,A 0.000,B 0.000,C 90.000,E1 50.723} C_DIS
LIN {X -0.165,Y -465.267,Z 519.075,A 0.000,B 0.000,C 90.000,E1 49.461} C_DIS
LIN {X 0.114,Y -466.742,Z 519.068,A 0.000,B 0.000,C 90.000,E1 48.162} C_DIS
LIN {X 0.003,Y -467.716,Z 519.062,A 0.000,B 0.000,C 90.000,E1 47.229} C_DIS
LIN {X -0.099,Y -468.523,Z 519.057,A 0.000,B 0.000,C 90.000,E1 46.296} C_DIS
LIN {X 0.132,Y -469.177,Z 519.052,A 0.000,B 0.000,C 90.000,E1 45.324} C_DIS
LIN {X 0.038,Y -469.692,Z 519.047,A 0.000,B 0.000,C 90.000,E1 44.393} C_DIS
LIN {X -0.047,Y -470.048,Z 519.041,A 0.000,B 0.000,C 90.000,E1 43.461} C_DIS
LIN {X -0.279,Y -470.256,Z 519.033,A 0.000,B 0.000,C 90.000,E1 41.919} C_DIS
LIN {X 0.079,Y -470.112,Z 519.026,A 0.000,B 0.000,C 90.000,E1 40.620} C_DIS
LIN {X 0.129,Y -469.794,Z 519.019,A 0.000,B 0.000,C 90.000,E1 39.358} C_DIS
LIN {X 0.175,Y -469.322,Z 519.012,A 0.000,B 0.000,C 90.000,E1 38.096} C_DIS
LIN {X -0.080,Y -468.780,Z 519.005,A 0.000,B 0.000,C 90.000,E1 36.870} C_DIS
LIN {X -0.047,Y -467.783,Z 518.994,A 0.000,B 0.000,C 90.000,E1 34.978} C_DIS
LIN {X 0.048,Y -467.071,Z 518.987,A 0.000,B 0.000,C 90.000,E1 33.706} C_DIS
LIN {X 0.162,Y -465.858,Z 518.977,A 0.000,B 0.000,C 90.000,E1 31.799} C_DIS
LIN {X 0.112,Y -465.029,Z 518.970,A 0.000,B 0.000,C 90.000,E1 30.541} C_DIS
LIN {X 0.054,Y -464.133,Z 518.963,A 0.000,B 0.000,C 90.000,E1 29.283} C_DIS
LIN {X -0.057,Y -462.530,Z 518.950,A 0.000,B 0.000,C 90.000,E1 27.078} C_DIS
LIN {X -0.004,Y -461.037,Z 518.938,A 0.000,B 0.000,C 90.000,E1 24.847} C_DIS
LIN {X -0.029,Y -460.133,Z 518.929,A 0.000,B 0.000,C 90.000,E1 23.259} C_DIS
LIN {X -0.263,Y -458.932,Z 518.915,A 0.000,B 0.000,C 90.000,E1 20.737} C_DIS
LIN {X 0.074,Y -458.205,Z 518.904,A 0.000,B 0.000,C 90.000,E1 18.779} C_DIS
LIN {X 0.100,Y -457.354,Z 518.888,A 0.000,B 0.000,C 90.000,E1 15.898} C_DIS
LIN {X 0.185,Y -457.065,Z 518.876,A 0.000,B 0.000,C 90.000,E1 13.647} C_DIS
LIN {X -0.165,Y -457.228,Z 518.862,A 0.000,B 0.000,C 90.000,E1 11.130} C_DIS
LIN {X 0.079,Y -457.639,Z 518.849,A 0.000,B 0.000,C 90.000,E1 8.859} C_DIS
LIN {X -0.028,Y -458.521,Z 518.835,A 0.000,B 0.000,C 90.000,E1 6.315} C_DIS
LIN {X -0.015,Y -460.065,Z 518.819,A 0.000,B 0.000,C 90.000,E1 3.440} C_DIS
LIN {X -0.155,Y -461.406,Z 518.809,A 0.000,B 0.000,C 90.000,E1 1.547} C_DIS
LIN {X 0.138,Y -463.457,Z 518.795,A 0.000,B 0.000,C 90.000,E1 359.141} C_DIS
LIN {X 0.063,Y -466.298,Z 518.781,A 0.000,B 0.000,C 90.000,E1 356.617} C_DIS
LIN {X -0.092,Y -469.877,Z 518.766,A 0.000,B 0.000,C 90.000,E1 353.799} C_DIS
LIN {X 0.210,Y -473.282,Z 518.752,A 0.000,B 0.000,C 90.000,E1 351.254} C_DIS
LIN {X -0.091,Y -476.349,Z 518.739,A 0.000,B 0.000,C 90.000,E1 349.106} C_DIS
LIN {X 0.183,Y -480.212,Z 518.726,A 0.000,B 0.000,C 90.000,E1 346.589} C_DIS
LIN {X -0.130,Y -484.765,Z 518.712,A 0.000,B 0.000,C 90.000,E1 344.157} C_DIS
LIN {X -0.062,Y -488.472,Z 518.702,A 0.000,B 0.000,C 90.000,E1 342.308} C_DIS
LIN {X -0.101,Y -491.612,Z 518.693,A 0.000,B 0.000,C 90.000,E1 340.786} C_DIS
LIN {X -0.028,Y -495.319,Z 518.683,A 0.000,B 0.000,C 90.000,E1 338.954} C_DIS
LIN {X 0.247,Y -498.430,Z 518.675,A 0.000,B 0.000,C 90.000,E1 337.411} C_DIS
LIN {X 0.116,Y -501.441,Z 518.666,A 0.000,B 0.000,C 90.000,E1 335.921} C_DIS
LIN {X 0.239,Y -504.342,Z 518.658,A 0.000,B 0.000,C 90.000,E1 334.409} C_DIS
LIN {X -0.098,Y -508.366,Z 518.646,A 0.000,B 0.000,C 90.000,E1 332.359} C_DIS
LIN {X 0.166,Y -511.201,Z 518.638,A 0.000,B 0.000,C 90.000,E1 330.845} C_DIS
LIN {X 0.049,Y -515.289,Z 518.627,A 0.000,B 0.000,C 90.000,E1 328.791} C_DIS
LIN {X -0.072,Y -518.835,Z 518.617,A 0.000,B 0.000,C 90.000,E1 327.041} C_DIS
LIN {X 0.157,Y -522.368,Z 518.607,A 0.000,B 0.000,C 90.000,E1 325.261} C_DIS
LIN {X -0.055,Y -525.343,Z 518.599,A 0.000,B 0.000,C 90.000,E1 323.829} C_DIS
LIN {X -0.235,Y -528.896,Z 518.589,A 0.000,B 0.000,C 90.000,E1 322.110} C_DIS
LIN {X 0.000,Y -531.846,Z 518.581,A 0.000,B 0.000,C 90.000,E1 320.642} C_DIS
LIN {X -0.130,Y -535.361,Z 518.572,A 0.000,B 0.000,C 90.000,E1 318.933} C_DIS
LIN {X 0.160,Y -538.361,Z 518.564,A 0.000,B 0.000,C 90.000,E1 317.472} C_DIS
LIN {X -0.265,Y -540.757,Z 518.558,A 0.000,B 0.000,C 90.000,E1 316.377} C_DIS
LIN {X -0.278,Y -544.234,Z 518.548,A 0.000,B 0.000,C 90.000,E1 314.676} C_DIS
LIN {X -0.193,Y -548.110,Z 518.537,A 0.000,B 0.000,C 90.000,E1 312.690} C_DIS
LIN {X -0.277,Y -553.566,Z 518.523,A 0.000,B 0.000,C 90.000,E1 310.172} C_DIS
LIN {X 0.067,Y -557.258,Z 518.514,A 0.000,B 0.000,C 90.000,E1 308.463} C_DIS
LIN {X -0.040,Y -559.465,Z 518.508,A 0.000,B 0.000,C 90.000,E1 307.363} C_DIS
LIN {X -0.165,Y -563.229,Z 518.497,A 0.000,B 0.000,C 90.000,E1 305.438} C_DIS
LIN {X -0.189,Y -571.146,Z 518.478,A 0.000,B 0.000,C 90.000,E1 302.005} C_DIS
LIN {X -0.281,Y -571.670,Z 518.477,A 0.000,B 0.000,C 90.000,E1 301.878} C_DIS
LIN {X -0.333,Y -573.263,Z 518.474,A 0.000,B 0.000,C 90.000,E1 301.337} C_DIS
LIN {X -0.081,Y -575.133,Z 518.471,A 0.000,B 0.000,C 90.000,E1 300.846} C_DIS
LIN {X -0.247,Y -575.900,Z 518.470,A 0.000,B 0.000,C 90.000,E1 300.590} C_DIS
LIN {X 0.227,Y -578.210,Z 518.467,A 0.000,B 0.000,C 90.000,E1 300.001} C_DIS
LIN {X 0.075,Y -579.740,Z 518.465,A 0.000,B 0.000,C 90.000,E1 299.745} C_DIS
LIN {X 0.145,Y -581.355,Z 518.463,A 0.000,B 0.000,C 90.000,E1 299.333} C_DIS
LIN {X -0.043,Y -585.968,Z 518.458,A 0.000,B 0.000,C 90.000,E1 298.409} C_DIS
LIN {X 0.123,Y -589.816,Z 518.453,A 0.000,B 0.000,C 90.000,E1 297.590} C_DIS
LIN {X 0.014,Y -590.867,Z 518.452,A 0.000,B 0.000,C 90.000,E1 297.334} C_DIS
LIN {X 0.075,Y -592.556,Z 518.449,A 0.000,B 0.000,C 90.000,E1 296.796} C_DIS
LIN {X 0.312,Y -594.199,Z 518.445,A 0.000,B 0.000,C 90.000,E1 295.976} C_DIS
LIN {X 0.125,Y -594.521,Z 518.442,A 0.000,B 0.000,C 90.000,E1 295.463} C_DIS
LIN {X 0.033,Y -594.561,Z 518.440,A 0.000,B 0.000,C 90.000,E1 295.207} C_DIS
LIN {X -0.152,Y -593.106,Z 518.437,A 0.000,B 0.000,C 90.000,E1 294.695} C_DIS
LIN {X 0.292,Y -592.077,Z 518.436,A 0.000,B 0.000,C 90.000,E1 294.387} C_DIS
LIN {X -0.099,Y -590.009,Z 518.433,A 0.000,B 0.000,C 90.000,E1 294.027} C_DIS
LIN {X -0.150,Y -589.176,Z 518.433,A 0.000,B 0.000,C 90.000,E1 293.898} C_DIS
LIN {X -0.203,Y -587.853,Z 518.432,A 0.000,B 0.000,C 90.000,E1 293.770} C_DIS
LIN {X 0.165,Y -584.505,Z 518.430,A 0.000,B 0.000,C 90.000,E1 293.334} C_DIS
LIN {X -0.028,Y -583.117,Z 518.429,A 0.000,B 0.000,C 90.000,E1 293.153} C_DIS
LIN {X -0.155,Y -581.780,Z 518.427,A 0.000,B 0.000,C 90.000,E1 292.898} C_DIS
LIN {X 0.056,Y -581.494,Z 518.427,A 0.000,B 0.000,C 90.000,E1 292.770} C_DIS
LIN {X 0.126,Y -581.112,Z 518.424,A 0.000,B 0.000,C 90.000,E1 292.386} C_DIS
LIN {X 0.089,Y -581.051,Z 518.420,A 0.000,B 0.000,C 90.000,E1 291.589} C_DIS
LIN {X -0.124,Y -581.818,Z 518.411,A 0.000,B 0.000,C 90.000,E1 289.993} C_DIS
LIN {X -0.024,Y -582.099,Z 518.405,A 0.000,B 0.000,C 90.000,E1 288.906} C_DIS
LIN {X -0.257,Y -582.248,Z 518.398,A 0.000,B 0.000,C 90.000,E1 287.583} C_DIS
LIN {X 0.072,Y -582.123,Z 518.390,A 0.000,B 0.000,C 90.000,E1 286.205} C_DIS
LIN {X 0.280,Y -581.742,Z 518.380,A 0.000,B 0.000,C 90.000,E1 284.300} C_DIS
LIN {X 0.324,Y -581.372,Z 518.369,A 0.000,B 0.000,C 90.000,E1 282.411} C_DIS
LIN {X 0.107,Y -580.802,Z 518.359,A 0.000,B 0.000,C 90.000,E1 280.546} C_DIS
LIN {X 0.227,Y -580.340,Z 518.350,A 0.000,B 0.000,C 90.000,E1 278.916} C_DIS
LIN {X -0.188,Y -579.721,Z 518.339,A 0.000,B 0.000,C 90.000,E1 277.068} C_DIS
LIN {X 0.175,Y -579.190,Z 518.332,A 0.000,B 0.000,C 90.000,E1 275.682} C_DIS
LIN {X 0.047,Y -578.350,Z 518.323,A 0.000,B 0.000,C 90.000,E1 274.073} C_DIS
LIN {X -0.257,Y -577.388,Z 518.315,A 0.000,B 0.000,C 90.000,E1 272.751} C_DIS
LIN {X -0.037,Y -576.298,Z 518.308,A 0.000,B 0.000,C 90.000,E1 271.375} C_DIS
LIN {X -0.002,Y -575.392,Z 518.302,A 0.000,B 0.000,C 90.000,E1 270.286} C_DIS
LIN {X 0.169,Y -574.017,Z 518.294,A 0.000,B 0.000,C 90.000,E1 268.912} C_DIS
LIN {X 0.188,Y -572.919,Z 518.288,A 0.000,B 0.000,C 90.000,E1 267.822} C_DIS
LIN {X 0.059,Y -570.961,Z 518.277,A 0.000,B 0.000,C 90.000,E1 265.927} C_DIS
LIN {X -0.244,Y -569.134,Z 518.268,A 0.000,B 0.000,C 90.000,E1 264.318} C_DIS
LIN {X -0.075,Y -567.489,Z 518.261,A 0.000,B 0.000,C 90.000,E1 262.932} C_DIS
LIN {X 0.065,Y -565.620,Z 518.253,A 0.000,B 0.000,C 90.000,E1 261.546} C_DIS
LIN {X -0.238,Y -563.276,Z 518.244,A 0.000,B 0.000,C 90.000,E1 259.926} C_DIS
LIN {X -0.152,Y -561.769,Z 518.238,A 0.000,B 0.000,C 90.000,E1 258.814} C_DIS
LIN {X 0.066,Y -559.696,Z 518.230,A 0.000,B 0.000,C 90.000,E1 257.409} C_DIS
LIN {X -0.171,Y -557.481,Z 518.222,A 0.000,B 0.000,C 90.000,E1 256.047} C_DIS
LIN {X 0.098,Y -555.030,Z 518.215,A 0.000,B 0.000,C 90.000,E1 254.629} C_DIS
LIN {X 0.194,Y -552.947,Z 518.208,A 0.000,B 0.000,C 90.000,E1 253.504} C_DIS
LIN {X -0.111,Y -550.661,Z 518.202,A 0.000,B 0.000,C 90.000,E1 252.417} C_DIS
LIN {X 0.079,Y -548.192,Z 518.196,A 0.000,B 0.000,C 90.000,E1 251.275} C_DIS
LIN {X -0.290,Y -545.693,Z 518.190,A 0.000,B 0.000,C 90.000,E1 250.188} C_DIS
LIN {X 0.240,Y -542.318,Z 518.182,A 0.000,B 0.000,C 90.000,E1 248.720} C_DIS
LIN {X -0.029,Y -539.485,Z 518.176,A 0.000,B 0.000,C 90.000,E1 247.614} C_DIS
LIN {X -0.130,Y -536.507,Z 518.169,A 0.000,B 0.000,C 90.000,E1 246.485} C_DIS
LIN {X -0.070,Y -532.606,Z 518.161,A 0.000,B 0.000,C 90.000,E1 245.049} C_DIS
LIN {X 0.136,Y -528.547,Z 518.153,A 0.000,B 0.000,C 90.000,E1 243.589} C_DIS
LIN {X 0.036,Y -524.324,Z 518.145,A 0.000,B 0.000,C 90.000,E1 242.153} C_DIS
LIN {X -0.003,Y -519.193,Z 518.136,A 0.000,B 0.000,C 90.000,E1 240.411} C_DIS
LIN {X -0.013,Y -514.850,Z 518.128,A 0.000,B 0.000,C 90.000,E1 238.948} C_DIS
LIN {X -0.178,Y -511.155,Z 518.121,A 0.000,B 0.000,C 90.000,E1 237.788} C_DIS
LIN {X -0.066,Y -506.478,Z 518.113,A 0.000,B 0.000,C 90.000,E1 236.294} C_DIS
LIN {X -0.117,Y -498.987,Z 518.099,A 0.000,B 0.000,C 90.000,E1 233.909} C_DIS
LIN {X 0.043,Y -492.916,Z 518.088,A 0.000,B 0.000,C 90.000,E1 231.778} C_DIS
LIN {X -0.100,Y -488.750,Z 518.079,A 0.000,B 0.000,C 90.000,E1 230.275} C_DIS
LIN {X 0.054,Y -484.527,Z 518.071,A 0.000,B 0.000,C 90.000,E1 228.728} C_DIS
LIN {X -0.153,Y -479.763,Z 518.061,A 0.000,B 0.000,C 90.000,E1 226.905} C_DIS
LIN {X 0.220,Y -474.969,Z 518.050,A 0.000,B 0.000,C 90.000,E1 225.000} C_DIS
LIN {X 0.135,Y -470.327,Z 518.040,A 0.000,B 0.000,C 90.000,E1 223.137} C_DIS
LIN {X 0.126,Y -464.447,Z 518.026,A 0.000,B 0.000,C 90.000,E1 220.620} C_DIS
LIN {X 0.257,Y -459.445,Z 518.013,A 0.000,B 0.000,C 90.000,E1 218.382} C_DIS
LIN {X 0.225,Y -456.005,Z 518.005,A 0.000,B 0.000,C 90.000,E1 216.790} C_DIS
LIN {X 0.033,Y -451.293,Z 517.992,A 0.000,B 0.000,C 90.000,E1 214.565} C_DIS
LIN {X 0.098,Y -446.841,Z 517.979,A 0.000,B 0.000,C 90.000,E1 212.291} C_DIS
LIN {X 0.171,Y -442.545,Z 517.967,A 0.000,B 0.000,C 90.000,E1 210.001} C_DIS
LIN {X 0.198,Y -439.613,Z 517.958,A 0.000,B 0.000,C 90.000,E1 208.359} C_DIS
LIN {X -0.017,Y -436.126,Z 517.947,A 0.000,B 0.000,C 90.000,E1 206.411} C_DIS
LIN {X 0.270,Y -432.786,Z 517.936,A 0.000,B 0.000,C 90.000,E1 204.387} C_DIS
LIN {X 0.107,Y -428.954,Z 517.923,A 0.000,B 0.000,C 90.000,E1 202.078} C_DIS
LIN {X 0.121,Y -425.035,Z 517.908,A 0.000,B 0.000,C 90.000,E1 199.396} C_DIS
LIN {X -0.124,Y -421.415,Z 517.893,A 0.000,B 0.000,C 90.000,E1 196.732} C_DIS
LIN {X -0.069,Y -419.775,Z 517.885,A 0.000,B 0.000,C 90.000,E1 195.371} C_DIS
LIN {X 0.174,Y -417.292,Z 517.874,A 0.000,B 0.000,C 90.000,E1 193.300} C_DIS
LIN {X 0.205,Y -415.296,Z 517.865,A 0.000,B 0.000,C 90.000,E1 191.591} C_DIS
LIN {X 0.031,Y -413.517,Z 517.855,A 0.000,B 0.000,C 90.000,E1 189.905} C_DIS
LIN {X -0.165,Y -411.047,Z 517.842,A 0.000,B 0.000,C 90.000,E1 187.530} C_DIS
LIN {X -0.075,Y -409.159,Z 517.832,A 0.000,B 0.000,C 90.000,E1 185.796} C_DIS
LIN {X -0.196,Y -405.489,Z 517.809,A 0.000,B 0.000,C 90.000,E1 181.661} C_DIS
LIN {X 0.049,Y -404.153,Z 517.798,A 0.000,B 0.000,C 90.000,E1 179.542} C_DIS
LIN {X 0.067,Y -402.200,Z 517.772,A 0.000,B 0.000,C 90.000,E1 175.008} C_DIS
LIN {X -0.126,Y -401.794,Z 517.759,A 0.000,B 0.000,C 90.000,E1 172.591} C_DIS
LIN {X -0.176,Y -401.800,Z 517.743,A 0.000,B 0.000,C 90.000,E1 169.803} C_DIS
LIN {X 0.007,Y -402.344,Z 517.724,A 0.000,B 0.000,C 90.000,E1 166.284} C_DIS
LIN {X -0.150,Y -403.013,Z 517.712,A 0.000,B 0.000,C 90.000,E1 164.212} C_DIS
LIN {X -0.092,Y -404.087,Z 517.699,A 0.000,B 0.000,C 90.000,E1 161.764} C_DIS
LIN {X -0.144,Y -405.497,Z 517.685,A 0.000,B 0.000,C 90.000,E1 159.337} C_DIS
LIN {X 0.123,Y -407.601,Z 517.668,A 0.000,B 0.000,C 90.000,E1 156.177} C_DIS
LIN {X 0.042,Y -409.520,Z 517.654,A 0.000,B 0.000,C 90.000,E1 153.768} C_DIS
LIN {X -0.109,Y -410.604,Z 517.647,A 0.000,B 0.000,C 90.000,E1 152.410} C_DIS
LIN {X -0.028,Y -412.127,Z 517.635,A 0.000,B 0.000,C 90.000,E1 150.333} C_DIS
LIN {X -0.076,Y -413.457,Z 517.624,A 0.000,B 0.000,C 90.000,E1 148.280} C_DIS
LIN {X 0.056,Y -414.460,Z 517.614,A 0.000,B 0.000,C 90.000,E1 146.548} C_DIS
LIN {X -0.021,Y -415.363,Z 517.605,A 0.000,B 0.000,C 90.000,E1 144.848} C_DIS
LIN {X 0.053,Y -416.223,Z 517.595,A 0.000,B 0.000,C 90.000,E1 143.130} C_DIS
LIN {X -0.042,Y -416.813,Z 517.588,A 0.000,B 0.000,C 90.000,E1 141.778} C_DIS
LIN {X -0.011,Y -417.414,Z 517.578,A 0.000,B 0.000,C 90.000,E1 140.070} C_DIS
LIN {X 0.184,Y -418.035,Z 517.567,A 0.000,B 0.000,C 90.000,E1 138.000} C_DIS
LIN {X 0.203,Y -418.323,Z 517.557,A 0.000,B 0.000,C 90.000,E1 136.296} C_DIS
LIN {X 0.212,Y -418.396,Z 517.548,A 0.000,B 0.000,C 90.000,E1 134.595} C_DIS
LIN {X 0.049,Y -418.291,Z 517.540,A 0.000,B 0.000,C 90.000,E1 133.257} C_DIS
LIN {X -0.117,Y -417.987,Z 517.533,A 0.000,B 0.000,C 90.000,E1 131.919} C_DIS
LIN {X 0.019,Y -417.315,Z 517.525,A 0.000,B 0.000,C 90.000,E1 130.539} C_DIS
LIN {X 0.060,Y -416.164,Z 517.516,A 0.000,B 0.000,C 90.000,E1 128.830} C_DIS
LIN {X -0.184,Y -414.938,Z 517.506,A 0.000,B 0.000,C 90.000,E1 127.156} C_DIS
LIN {X -0.189,Y -414.372,Z 517.502,A 0.000,B 0.000,C 90.000,E1 126.377} C_DIS
LIN {X -0.228,Y -414.380,Z 517.502,A 0.000,B 0.000,C 90.000,E1 126.377} C_DIS
LIN {X 0.038,Y -416.033,Z 517.499,A 0.000,B 0.000,C 90.000,E1 125.758} C_DIS
LIN {X 0.167,Y -425.545,Z 517.478,A 0.000,B 0.000,C 90.000,E1 122.005} C_DIS
LIN {X 0.111,Y -430.577,Z 517.469,A 0.000,B 0.000,C 90.000,E1 120.335} C_DIS
LIN {X -0.088,Y -441.486,Z 517.445,A 0.000,B 0.000,C 90.000,E1 116.052} C_DIS
LIN {X -0.170,Y -444.400,Z 517.439,A 0.000,B 0.000,C 90.000,E1 115.079} C_DIS
LIN {X 0.088,Y -445.210,Z 517.437,A 0.000,B 0.000,C 90.000,E1 114.719} C_DIS
LIN {X -0.049,Y -454.409,Z 517.416,A 0.000,B 0.000,C 90.000,E1 110.844} C_DIS
LIN {X -0.034,Y -455.685,Z 517.413,A 0.000,B 0.000,C 90.000,E1 110.375} C_DIS
LIN {X -0.074,Y -455.709,Z 517.413,A 0.000,B 0.000,C 90.000,E1 110.375} C_DIS
LIN {X -0.145,Y -482.223,Z 517.408,A 0.000,B 0.000,C 90.000,E1 109.504} C_DIS
LIN {X -0.003,Y -492.657,Z 517.406,A 0.000,B 0.000,C 90.000,E1 109.141} C_DIS
LIN {X -0.079,Y -503.059,Z 517.404,A 0.000,B 0.000,C 90.000,E1 108.779} C_DIS
LIN {X 0.172,Y -516.925,Z 517.401,A 0.000,B 0.000,C 90.000,E1 108.236} C_DIS
LIN {X -0.151,Y -527.228,Z 517.399,A 0.000,B 0.000,C 90.000,E1 107.873} C_DIS
LIN {X -0.163,Y -537.387,Z 517.397,A 0.000,B 0.000,C 90.000,E1 107.457} C_DIS
LIN {X -0.060,Y -543.930,Z 517.395,A 0.000,B 0.000,C 90.000,E1 107.149} C_DIS
LIN {X 0.177,Y -550.342,Z 517.393,A 0.000,B 0.000,C 90.000,E1 106.804} C_DIS
LIN {X -0.197,Y -556.696,Z 517.392,A 0.000,B 0.000,C 90.000,E1 106.496} C_DIS
LIN {X -0.241,Y -559.929,Z 517.391,A 0.000,B 0.000,C 90.000,E1 106.315} C_DIS
LIN {X 0.145,Y -565.712,Z 517.388,A 0.000,B 0.000,C 90.000,E1 105.898} C_DIS
LIN {X 0.108,Y -571.628,Z 517.386,A 0.000,B 0.000,C 90.000,E1 105.481} C_DIS
LIN {X -0.186,Y -577.315,Z 517.384,A 0.000,B 0.000,C 90.000,E1 105.064} C_DIS
LIN {X -0.165,Y -582.755,Z 517.381,A 0.000,B 0.000,C 90.000,E1 104.592} C_DIS
LIN {X 0.109,Y -588.627,Z 517.378,A 0.000,B 0.000,C 90.000,E1 104.008} C_DIS
LIN {X -0.072,Y -594.459,Z 517.375,A 0.000,B 0.000,C 90.000,E1 103.411} C_DIS
LIN {X 0.051,Y -597.816,Z 517.372,A 0.000,B 0.000,C 90.000,E1 103.008} C_DIS
LIN {X 0.088,Y -602.461,Z 517.369,A 0.000,B 0.000,C 90.000,E1 102.479} C_DIS
LIN {X -0.211,Y -609.873,Z 517.364,A 0.000,B 0.000,C 90.000,E1 101.591} C_DIS
LIN {X -0.182,Y -616.288,Z 517.359,A 0.000,B 0.000,C 90.000,E1 100.715} C_DIS
LIN {X -0.230,Y -620.726,Z 517.356,A 0.000,B 0.000,C 90.000,E1 100.074} C_DIS
LIN {X -0.238,Y -624.901,Z 517.352,A 0.000,B 0.000,C 90.000,E1 99.434} C_DIS
LIN {X 0.251,Y -629.398,Z 517.348,A 0.000,B 0.000,C 90.000,E1 98.624} C_DIS
LIN {X -0.305,Y -633.462,Z 517.344,A 0.000,B 0.000,C 90.000,E1 97.936} C_DIS
LIN {X 0.092,Y -638.730,Z 517.338,A 0.000,B 0.000,C 90.000,E1 96.891} C_DIS
LIN {X 0.150,Y -641.787,Z 517.335,A 0.000,B 0.000,C 90.000,E1 96.258} C_DIS
LIN {X -0.065,Y -646.296,Z 517.329,A 0.000,B 0.000,C 90.000,E1 95.277} C_DIS
LIN {X -0.061,Y -649.478,Z 517.325,A 0.000,B 0.000,C 90.000,E1 94.531} C_DIS
LIN {X -0.237,Y -653.243,Z 517.320,A 0.000,B 0.000,C 90.000,E1 93.555} C_DIS
LIN {X -0.164,Y -655.545,Z 517.316,A 0.000,B 0.000,C 90.000,E1 92.808} C_DIS
LIN {X 0.095,Y -656.928,Z 517.313,A 0.000,B 0.000,C 90.000,E1 92.293} C_DIS
LIN {X -0.268,Y -658.087,Z 517.310,A 0.000,B 0.000,C 90.000,E1 91.833} C_DIS
LIN {X -0.175,Y -659.386,Z 517.306,A 0.000,B 0.000,C 90.000,E1 91.088} C_DIS
LIN {X 0.116,Y -659.991,Z 517.303,A 0.000,B 0.000,C 90.000,E1 90.573} C_DIS
LIN {X -0.247,Y -660.444,Z 517.301,A 0.000,B 0.000,C 90.000,E1 90.115} C_DIS
LIN {X 0.054,Y -660.594,Z 517.298,A 0.000,B 0.000,C 90.000,E1 89.599} C_DIS
LIN {X 0.176,Y -660.496,Z 517.294,A 0.000,B 0.000,C 90.000,E1 88.854} C_DIS
LIN {X -0.185,Y -660.300,Z 517.291,A 0.000,B 0.000,C 90.000,E1 88.396} C_DIS
LIN {X 0.133,Y -659.828,Z 517.288,A 0.000,B 0.000,C 90.000,E1 87.879} C_DIS
LIN {X 0.241,Y -658.804,Z 517.284,A 0.000,B 0.000,C 90.000,E1 87.135} C_DIS
LIN {X -0.287,Y -657.405,Z 517.280,A 0.000,B 0.000,C 90.000,E1 86.445} C_DIS
LIN {X 0.176,Y -656.923,Z 517.279,A 0.000,B 0.000,C 90.000,E1 86.159} C_DIS
LIN {X -0.168,Y -655.760,Z 517.276,A 0.000,B 0.000,C 90.000,E1 85.698} C_DIS
LIN {X -0.067,Y -653.657,Z 517.272,A 0.000,B 0.000,C 90.000,E1 84.951} C_DIS
LIN {X 0.011,Y -651.075,Z 517.268,A 0.000,B 0.000,C 90.000,E1 84.204} C_DIS
LIN {X 0.133,Y -648.372,Z 517.264,A 0.000,B 0.000,C 90.000,E1 83.451} C_DIS
LIN {X 0.152,Y -645.306,Z 517.260,A 0.000,B 0.000,C 90.000,E1 82.704} C_DIS
LIN {X 0.092,Y -641.125,Z 517.255,A 0.000,B 0.000,C 90.000,E1 81.837} C_DIS
LIN {X 0.253,Y -637.956,Z 517.251,A 0.000,B 0.000,C 90.000,E1 81.197} C_DIS
LIN {X -0.201,Y -635.291,Z 517.248,A 0.000,B 0.000,C 90.000,E1 80.735} C_DIS
LIN {X -0.238,Y -630.872,Z 517.244,A 0.000,B 0.000,C 90.000,E1 79.982} C_DIS
LIN {X -0.165,Y -626.958,Z 517.241,A 0.000,B 0.000,C 90.000,E1 79.342} C_DIS
LIN {X -0.126,Y -622.856,Z 517.237,A 0.000,B 0.000,C 90.000,E1 78.701} C_DIS
LIN {X -0.173,Y -617.563,Z 517.233,A 0.000,B 0.000,C 90.000,E1 77.937} C_DIS
LIN {X -0.269,Y -611.668,Z 517.229,A 0.000,B 0.000,C 90.000,E1 77.173} C_DIS
LIN {X 0.115,Y -606.418,Z 517.225,A 0.000,B 0.000,C 90.000,E1 76.520} C_DIS
LIN {X 0.114,Y -600.329,Z 517.222,A 0.000,B 0.000,C 90.000,E1 75.880} C_DIS
LIN {X -0.127,Y -596.524,Z 517.220,A 0.000,B 0.000,C 90.000,E1 75.519} C_DIS
LIN {X 0.233,Y -589.713,Z 517.216,A 0.000,B 0.000,C 90.000,E1 74.866} C_DIS
LIN {X 0.148,Y -585.539,Z 517.214,A 0.000,B 0.000,C 90.000,E1 74.519} C_DIS
LIN {X -0.188,Y -579.672,Z 517.212,A 0.000,B 0.000,C 90.000,E1 74.102} C_DIS
LIN {X -0.264,Y -573.556,Z 517.209,A 0.000,B 0.000,C 90.000,E1 73.685} C_DIS
LIN {X -0.210,Y -568.828,Z 517.208,A 0.000,B 0.000,C 90.000,E1 73.378} C_DIS
LIN {X 0.152,Y -562.084,Z 517.205,A 0.000,B 0.000,C 90.000,E1 72.960} C_DIS
LIN {X -0.105,Y -556.956,Z 517.204,A 0.000,B 0.000,C 90.000,E1 72.725} C_DIS
LIN {X -0.192,Y -549.961,Z 517.202,A 0.000,B 0.000,C 90.000,E1 72.417} C_DIS
LIN {X -0.065,Y -542.568,Z 517.201,A 0.000,B 0.000,C 90.000,E1 72.127} C_DIS
LIN {X -0.076,Y -538.931,Z 517.200,A 0.000,B 0.000,C 90.000,E1 72.000} C_DIS
LIN {X 0.046,Y -531.373,Z 517.199,A 0.000,B 0.000,C 90.000,E1 71.764} C_DIS
LIN {X -0.125,Y -525.680,Z 517.198,A 0.000,B 0.000,C 90.000,E1 71.638} C_DIS
LIN {X 0.044,Y -506.820,Z 517.196,A 0.000,B 0.000,C 90.000,E1 71.221} C_DIS
LIN {X 0.169,Y -501.016,Z 517.195,A 0.000,B 0.000,C 90.000,E1 71.094} C_DIS
LIN {X -0.093,Y -487.403,Z 517.194,A 0.000,B 0.000,C 90.000,E1 70.913} C_DIS
LIN {X -0.019,Y -471.508,Z 517.193,A 0.000,B 0.000,C 90.000,E1 70.678} C_DIS
LIN {X -0.050,Y -471.418,Z 517.193,A 0.000,B 0.000,C 90.000,E1 70.678} C_DIS
LIN {X -0.117,Y -465.789,Z 517.173,A 0.000,B 0.000,C 90.000,E1 67.177} C_DIS
LIN {X -0.054,Y -464.430,Z 517.170,A 0.000,B 0.000,C 90.000,E1 66.538} C_DIS
LIN {X -0.119,Y -456.278,Z 517.147,A 0.000,B 0.000,C 90.000,E1 62.410} C_DIS
LIN {X -0.120,Y -455.135,Z 517.143,A 0.000,B 0.000,C 90.000,E1 61.769} C_DIS
LIN {X -0.056,Y -446.682,Z 517.122,A 0.000,B 0.000,C 90.000,E1 57.995} C_DIS
LIN {X -0.096,Y -446.685,Z 517.122,A 0.000,B 0.000,C 90.000,E1 57.995} C_DIS
LIN {X -0.061,Y -450.204,Z 517.116,A 0.000,B 0.000,C 90.000,E1 56.914} C_DIS
LIN {X 0.056,Y -453.149,Z 517.111,A 0.000,B 0.000,C 90.000,E1 55.928} C_DIS
LIN {X 0.050,Y -456.726,Z 517.104,A 0.000,B 0.000,C 90.000,E1 54.642} C_DIS
LIN {X 0.251,Y -459.733,Z 517.097,A 0.000,B 0.000,C 90.000,E1 53.336} C_DIS
LIN {X 0.096,Y -461.109,Z 517.093,A 0.000,B 0.000,C 90.000,E1 52.718} C_DIS
LIN {X -0.137,Y -462.340,Z 517.089,A 0.000,B 0.000,C 90.000,E1 52.110} C_DIS
LIN {X 0.161,Y -464.362,Z 517.082,A 0.000,B 0.000,C 90.000,E1 50.803} C_DIS
LIN {X -0.286,Y -465.746,Z 517.077,A 0.000,B 0.000,C 90.000,E1 49.908} C_DIS
LIN {X -0.061,Y -466.919,Z 517.072,A 0.000,B 0.000,C 90.000,E1 48.933} C_DIS
LIN {X -0.101,Y -468.324,Z 517.065,A 0.000,B 0.000,C 90.000,E1 47.676} C_DIS
LIN {X 0.226,Y -469.391,Z 517.058,A 0.000,B 0.000,C 90.000,E1 46.377} C_DIS
LIN {X -0.197,Y -470.052,Z 517.053,A 0.000,B 0.000,C 90.000,E1 45.486} C_DIS
LIN {X 0.139,Y -470.654,Z 517.046,A 0.000,B 0.000,C 90.000,E1 44.190} C_DIS
LIN {X -0.016,Y -470.898,Z 517.042,A 0.000,B 0.000,C 90.000,E1 43.581} C_DIS
LIN {X 0.009,Y -471.060,Z 517.035,A 0.000,B 0.000,C 90.000,E1 42.324} C_DIS
LIN {X -0.053,Y -471.045,Z 517.030,A 0.000,B 0.000,C 90.000,E1 41.391} C_DIS
LIN {X -0.041,Y -470.807,Z 517.023,A 0.000,B 0.000,C 90.000,E1 40.135} C_DIS
LIN {X 0.153,Y -470.297,Z 517.014,A 0.000,B 0.000,C 90.000,E1 38.543} C_DIS
LIN {X -0.027,Y -469.579,Z 517.006,A 0.000,B 0.000,C 90.000,E1 36.996} C_DIS
LIN {X 0.017,Y -468.576,Z 516.995,A 0.000,B 0.000,C 90.000,E1 35.105} C_DIS
LIN {X 0.122,Y -467.842,Z 516.988,A 0.000,B 0.000,C 90.000,E1 33.833} C_DIS
LIN {X 0.100,Y -466.841,Z 516.979,A 0.000,B 0.000,C 90.000,E1 32.260} C_DIS
LIN {X 0.210,Y -465.774,Z 516.971,A 0.000,B 0.000,C 90.000,E1 30.669} C_DIS
LIN {X -0.102,Y -464.585,Z 516.962,A 0.000,B 0.000,C 90.000,E1 29.127} C_DIS
LIN {X 0.198,Y -462.947,Z 516.949,A 0.000,B 0.000,C 90.000,E1 26.873} C_DIS
LIN {X 0.136,Y -461.660,Z 516.939,A 0.000,B 0.000,C 90.000,E1 24.975} C_DIS
LIN {X 0.046,Y -460.505,Z 516.928,A 0.000,B 0.000,C 90.000,E1 23.078} C_DIS
LIN {X -0.091,Y -459.414,Z 516.916,A 0.000,B 0.000,C 90.000,E1 20.865} C_DIS
LIN {X -0.171,Y -458.681,Z 516.905,A 0.000,B 0.000,C 90.000,E1 18.960} C_DIS
LIN {X -0.128,Y -457.765,Z 516.889,A 0.000,B 0.000,C 90.000,E1 16.079} C_DIS
LIN {X -0.028,Y -457.442,Z 516.877,A 0.000,B 0.000,C 90.000,E1 13.828} C_DIS
LIN {X 0.175,Y -457.477,Z 516.863,A 0.000,B 0.000,C 90.000,E1 11.243} C_DIS
LIN {X 0.127,Y -457.959,Z 516.848,A 0.000,B 0.000,C 90.000,E1 8.690} C_DIS
LIN {X -0.190,Y -458.961,Z 516.832,A 0.000,B 0.000,C 90.000,E1 5.853} C_DIS
LIN {X -0.130,Y -460.150,Z 516.820,A 0.000,B 0.000,C 90.000,E1 3.612} C_DIS
LIN {X -0.065,Y -461.703,Z 516.808,A 0.000,B 0.000,C 90.000,E1 1.375} C_DIS
LIN {X -0.074,Y -463.336,Z 516.797,A 0.000,B 0.000,C 90.000,E1 359.484} C_DIS
LIN {X 0.069,Y -466.423,Z 516.781,A 0.000,B 0.000,C 90.000,E1 356.617} C_DIS
LIN {X -0.113,Y -469.160,Z 516.769,A 0.000,B 0.000,C 90.000,E1 354.432} C_DIS
LIN {X 0.240,Y -471.206,Z 516.760,A 0.000,B 0.000,C 90.000,E1 352.818} C_DIS
LIN {X -0.019,Y -473.818,Z 516.750,A 0.000,B 0.000,C 90.000,E1 350.971} C_DIS
LIN {X 0.079,Y -477.418,Z 516.736,A 0.000,B 0.000,C 90.000,E1 348.465} C_DIS
LIN {X 0.186,Y -483.154,Z 516.717,A 0.000,B 0.000,C 90.000,E1 345.046} C_DIS
LIN {X 0.103,Y -488.017,Z 516.703,A 0.000,B 0.000,C 90.000,E1 342.598} C_DIS
LIN {X -0.097,Y -491.177,Z 516.695,A 0.000,B 0.000,C 90.000,E1 341.094} C_DIS
LIN {X -0.037,Y -494.914,Z 516.685,A 0.000,B 0.000,C 90.000,E1 339.263} C_DIS
LIN {X 0.041,Y -498.030,Z 516.676,A 0.000,B 0.000,C 90.000,E1 337.741} C_DIS
LIN {X 0.163,Y -501.697,Z 516.666,A 0.000,B 0.000,C 90.000,E1 335.921} C_DIS
LIN {X -0.163,Y -504.591,Z 516.658,A 0.000,B 0.000,C 90.000,E1 334.460} C_DIS
LIN {X 0.013,Y -507.441,Z 516.650,A 0.000,B 0.000,C 90.000,E1 332.948} C_DIS
LIN {X -0.106,Y -510.951,Z 516.640,A 0.000,B 0.000,C 90.000,E1 331.179} C_DIS
LIN {X 0.123,Y -515.618,Z 516.627,A 0.000,B 0.000,C 90.000,E1 328.791} C_DIS
LIN {X 0.010,Y -519.213,Z 516.617,A 0.000,B 0.000,C 90.000,E1 327.041} C_DIS
LIN {X 0.157,Y -524.002,Z 516.604,A 0.000,B 0.000,C 90.000,E1 324.689} C_DIS
LIN {X -0.021,Y -526.962,Z 516.596,A 0.000,B 0.000,C 90.000,E1 323.256} C_DIS
LIN {X -0.147,Y -529.964,Z 516.588,A 0.000,B 0.000,C 90.000,E1 321.823} C_DIS
LIN {X 0.094,Y -533.522,Z 516.578,A 0.000,B 0.000,C 90.000,E1 320.070} C_DIS
LIN {X -0.005,Y -536.464,Z 516.570,A 0.000,B 0.000,C 90.000,E1 318.647} C_DIS
LIN {X -0.097,Y -540.120,Z 516.561,A 0.000,B 0.000,C 90.000,E1 316.944} C_DIS
LIN {X -0.127,Y -543.600,Z 516.551,A 0.000,B 0.000,C 90.000,E1 315.243} C_DIS
LIN {X 0.275,Y -545.292,Z 516.547,A 0.000,B 0.000,C 90.000,E1 314.352} C_DIS
LIN {X 0.018,Y -549.189,Z 516.536,A 0.000,B 0.000,C 90.000,E1 312.405} C_DIS
LIN {X -0.020,Y -554.632,Z 516.522,A 0.000,B 0.000,C 90.000,E1 309.886} C_DIS
LIN {X 0.271,Y -557.687,Z 516.514,A 0.000,B 0.000,C 90.000,E1 308.463} C_DIS
LIN {X 0.170,Y -559.897,Z 516.508,A 0.000,B 0.000,C 90.000,E1 307.363} C_DIS
LIN {X -0.044,Y -563.122,Z 516.498,A 0.000,B 0.000,C 90.000,E1 305.724} C_DIS
LIN {X 0.023,Y -570.272,Z 516.480,A 0.000,B 0.000,C 90.000,E1 302.418} C_DIS
LIN {X 0.084,Y -572.236,Z 516.476,A 0.000,B 0.000,C 90.000,E1 301.592} C_DIS
LIN {X 0.034,Y -573.572,Z 516.473,A 0.000,B 0.000,C 90.000,E1 301.052} C_DIS
LIN {X -0.092,Y -575.421,Z 516.469,A 0.000,B 0.000,C 90.000,E1 300.384} C_DIS
LIN {X -0.333,Y -577.109,Z 516.467,A 0.000,B 0.000,C 90.000,E1 300.001} C_DIS
LIN {X 0.300,Y -577.891,Z 516.465,A 0.000,B 0.000,C 90.000,E1 299.667} C_DIS
LIN {X 0.149,Y -578.940,Z 516.464,A 0.000,B 0.000,C 90.000,E1 299.411} C_DIS
LIN {X -0.071,Y -580.318,Z 516.461,A 0.000,B 0.000,C 90.000,E1 299.027} C_DIS
LIN {X -0.011,Y -581.924,Z 516.460,A 0.000,B 0.000,C 90.000,E1 298.743} C_DIS
LIN {X -0.149,Y -582.741,Z 516.458,A 0.000,B 0.000,C 90.000,E1 298.487} C_DIS
LIN {X -0.347,Y -584.437,Z 516.456,A 0.000,B 0.000,C 90.000,E1 298.103} C_DIS
LIN {X 0.105,Y -585.166,Z 516.455,A 0.000,B 0.000,C 90.000,E1 297.924} C_DIS
LIN {X 0.022,Y -586.867,Z 516.452,A 0.000,B 0.000,C 90.000,E1 297.436} C_DIS
LIN {X -0.097,Y -587.895,Z 516.451,A 0.000,B 0.000,C 90.000,E1 297.180} C_DIS
LIN {X 0.310,Y -588.782,Z 516.450,A 0.000,B 0.000,C 90.000,E1 296.873} C_DIS
LIN {X 0.088,Y -589.846,Z 516.447,A 0.000,B 0.000,C 90.000,E1 296.360} C_DIS
LIN {X -0.020,Y -590.269,Z 516.445,A 0.000,B 0.000,C 90.000,E1 296.104} C_DIS
LIN {X -0.232,Y -590.731,Z 516.442,A 0.000,B 0.000,C 90.000,E1 295.591} C_DIS
LIN {X 0.197,Y -590.642,Z 516.441,A 0.000,B 0.000,C 90.000,E1 295.283} C_DIS
LIN {X -0.010,Y -590.072,Z 516.438,A 0.000,B 0.000,C 90.000,E1 294.771} C_DIS
LIN {X -0.116,Y -589.370,Z 516.436,A 0.000,B 0.000,C 90.000,E1 294.515} C_DIS
LIN {X -0.224,Y -588.344,Z 516.435,A 0.000,B 0.000,C 90.000,E1 294.259} C_DIS
LIN {X 0.203,Y -587.148,Z 516.433,A 0.000,B 0.000,C 90.000,E1 293.951} C_DIS
LIN {X 0.088,Y -585.600,Z 516.432,A 0.000,B 0.000,C 90.000,E1 293.695} C_DIS
LIN {X 0.117,Y -583.285,Z 516.430,A 0.000,B 0.000,C 90.000,E1 293.387} C_DIS
LIN {X 0.075,Y -583.269,Z 516.430,A 0.000,B 0.000,C 90.000,E1 293.387} C_DIS
LIN {X 0.144,Y -582.924,Z 516.429,A 0.000,B 0.000,C 90.000,E1 293.153} C_DIS
LIN {X 0.079,Y -582.498,Z 516.428,A 0.000,B 0.000,C 90.000,E1 293.025} C_DIS
LIN {X -0.068,Y -582.139,Z 516.427,A 0.000,B 0.000,C 90.000,E1 292.770} C_DIS
LIN {X 0.194,Y -581.976,Z 516.424,A 0.000,B 0.000,C 90.000,E1 292.206} C_DIS
LIN {X 0.144,Y -582.388,Z 516.416,A 0.000,B 0.000,C 90.000,E1 290.865} C_DIS
LIN {X 0.054,Y -582.904,Z 516.412,A 0.000,B 0.000,C 90.000,E1 290.066} C_DIS
LIN {X 0.025,Y -583.237,Z 516.404,A 0.000,B 0.000,C 90.000,E1 288.725} C_DIS
LIN {X 0.148,Y -583.404,Z 516.398,A 0.000,B 0.000,C 90.000,E1 287.638} C_DIS
LIN {X -0.067,Y -583.340,Z 516.391,A 0.000,B 0.000,C 90.000,E1 286.315} C_DIS
LIN {X -0.171,Y -582.970,Z 516.379,A 0.000,B 0.000,C 90.000,E1 284.175} C_DIS
LIN {X 0.102,Y -582.717,Z 516.370,A 0.000,B 0.000,C 90.000,E1 282.535} C_DIS
LIN {X 0.037,Y -582.208,Z 516.359,A 0.000,B 0.000,C 90.000,E1 280.658} C_DIS
LIN {X -0.255,Y -581.686,Z 516.349,A 0.000,B 0.000,C 90.000,E1 278.803} C_DIS
LIN {X -0.206,Y -581.191,Z 516.340,A 0.000,B 0.000,C 90.000,E1 277.182} C_DIS
LIN {X 0.181,Y -580.684,Z 516.332,A 0.000,B 0.000,C 90.000,E1 275.796} C_DIS
LIN {X 0.081,Y -579.828,Z 516.323,A 0.000,B 0.000,C 90.000,E1 274.188} C_DIS
LIN {X -0.198,Y -578.886,Z 516.316,A 0.000,B 0.000,C 90.000,E1 272.865} C_DIS
LIN {X -0.113,Y -577.991,Z 516.310,A 0.000,B 0.000,C 90.000,E1 271.776} C_DIS
LIN {X 0.101,Y -576.842,Z 516.302,A 0.000,B 0.000,C 90.000,E1 270.401} C_DIS
LIN {X -0.127,Y -575.145,Z 516.293,A 0.000,B 0.000,C 90.000,E1 268.797} C_DIS
LIN {X -0.093,Y -573.973,Z 516.287,A 0.000,B 0.000,C 90.000,E1 267.707} C_DIS
LIN {X 0.201,Y -572.254,Z 516.278,A 0.000,B 0.000,C 90.000,E1 266.045} C_DIS
LIN {X 0.085,Y -570.032,Z 516.268,A 0.000,B 0.000,C 90.000,E1 264.147} C_DIS
LIN {X 0.265,Y -568.326,Z 516.260,A 0.000,B 0.000,C 90.000,E1 262.761} C_DIS
LIN {X -0.318,Y -566.813,Z 516.254,A 0.000,B 0.000,C 90.000,E1 261.724} C_DIS
LIN {X -0.175,Y -563.594,Z 516.242,A 0.000,B 0.000,C 90.000,E1 259.511} C_DIS
LIN {X -0.189,Y -561.986,Z 516.236,A 0.000,B 0.000,C 90.000,E1 258.409} C_DIS
LIN {X 0.151,Y -559.842,Z 516.228,A 0.000,B 0.000,C 90.000,E1 256.992} C_DIS
LIN {X -0.215,Y -557.536,Z 516.220,A 0.000,B 0.000,C 90.000,E1 255.644} C_DIS
LIN {X -0.219,Y -554.470,Z 516.211,A 0.000,B 0.000,C 90.000,E1 253.976} C_DIS
LIN {X 0.134,Y -551.612,Z 516.203,A 0.000,B 0.000,C 90.000,E1 252.543} C_DIS
LIN {X -0.186,Y -549.174,Z 516.197,A 0.000,B 0.000,C 90.000,E1 251.456} C_DIS
LIN {X 0.227,Y -545.994,Z 516.189,A 0.000,B 0.000,C 90.000,E1 250.007} C_DIS
LIN {X 0.252,Y -542.572,Z 516.181,A 0.000,B 0.000,C 90.000,E1 248.592} C_DIS
LIN {X -0.012,Y -539.655,Z 516.175,A 0.000,B 0.000,C 90.000,E1 247.486} C_DIS
LIN {X -0.109,Y -536.653,Z 516.169,A 0.000,B 0.000,C 90.000,E1 246.357} C_DIS
LIN {X -0.046,Y -532.689,Z 516.161,A 0.000,B 0.000,C 90.000,E1 244.921} C_DIS
LIN {X -0.015,Y -529.416,Z 516.154,A 0.000,B 0.000,C 90.000,E1 243.768} C_DIS
LIN {X 0.128,Y -525.202,Z 516.146,A 0.000,B 0.000,C 90.000,E1 242.308} C_DIS
LIN {X -0.103,Y -520.010,Z 516.137,A 0.000,B 0.000,C 90.000,E1 240.589} C_DIS
LIN {X -0.089,Y -515.700,Z 516.128,A 0.000,B 0.000,C 90.000,E1 239.125} C_DIS
LIN {X 0.200,Y -512.006,Z 516.122,A 0.000,B 0.000,C 90.000,E1 237.916} C_DIS
LIN {X 0.328,Y -507.318,Z 516.114,A 0.000,B 0.000,C 90.000,E1 236.421} C_DIS
LIN {X 0.125,Y -500.684,Z 516.102,A 0.000,B 0.000,C 90.000,E1 234.356} C_DIS
LIN {X -0.209,Y -493.609,Z 516.089,A 0.000,B 0.000,C 90.000,E1 231.984} C_DIS
LIN {X -0.117,Y -488.567,Z 516.079,A 0.000,B 0.000,C 90.000,E1 230.150} C_DIS
LIN {X 0.073,Y -481.955,Z 516.065,A 0.000,B 0.000,C 90.000,E1 227.676} C_DIS
LIN {X -0.069,Y -478.754,Z 516.058,A 0.000,B 0.000,C 90.000,E1 226.458} C_DIS
LIN {X -0.169,Y -474.778,Z 516.049,A 0.000,B 0.000,C 90.000,E1 224.919} C_DIS
LIN {X 0.000,Y -470.916,Z 516.041,A 0.000,B 0.000,C 90.000,E1 223.338} C_DIS
LIN {X -0.021,Y -464.997,Z 516.027,A 0.000,B 0.000,C 90.000,E1 220.825} C_DIS
LIN {X -0.167,Y -459.989,Z 516.015,A 0.000,B 0.000,C 90.000,E1 218.624} C_DIS
LIN {X 0.096,Y -456.538,Z 516.006,A 0.000,B 0.000,C 90.000,E1 216.996} C_DIS
LIN {X 0.173,Y -451.825,Z 515.993,A 0.000,B 0.000,C 90.000,E1 214.739} C_DIS
LIN {X -0.003,Y -447.385,Z 515.981,A 0.000,B 0.000,C 90.000,E1 212.498} C_DIS
LIN {X 0.089,Y -443.062,Z 515.968,A 0.000,B 0.000,C 90.000,E1 210.207} C_DIS
LIN {X 0.171,Y -439.522,Z 515.957,A 0.000,B 0.000,C 90.000,E1 208.231} C_DIS
LIN {X -0.068,Y -436.622,Z 515.948,A 0.000,B 0.000,C 90.000,E1 206.616} C_DIS
LIN {X -0.155,Y -433.254,Z 515.937,A 0.000,B 0.000,C 90.000,E1 204.643} C_DIS
LIN {X 0.077,Y -430.483,Z 515.928,A 0.000,B 0.000,C 90.000,E1 202.950} C_DIS
LIN {X 0.089,Y -426.825,Z 515.915,A 0.000,B 0.000,C 90.000,E1 200.610} C_DIS
LIN {X -0.128,Y -424.450,Z 515.905,A 0.000,B 0.000,C 90.000,E1 198.960} C_DIS
LIN {X 0.051,Y -421.741,Z 515.894,A 0.000,B 0.000,C 90.000,E1 196.913} C_DIS
LIN {X -0.126,Y -419.665,Z 515.885,A 0.000,B 0.000,C 90.000,E1 195.245} C_DIS
LIN {X 0.108,Y -417.199,Z 515.873,A 0.000,B 0.000,C 90.000,E1 193.175} C_DIS
LIN {X 0.146,Y -414.509,Z 515.860,A 0.000,B 0.000,C 90.000,E1 190.782} C_DIS
LIN {X -0.078,Y -413.063,Z 515.852,A 0.000,B 0.000,C 90.000,E1 189.443} C_DIS
LIN {X 0.147,Y -410.982,Z 515.841,A 0.000,B 0.000,C 90.000,E1 187.352} C_DIS
LIN {X 0.184,Y -408.404,Z 515.828,A 0.000,B 0.000,C 90.000,E1 184.935} C_DIS
LIN {X 0.014,Y -404.991,Z 515.805,A 0.000,B 0.000,C 90.000,E1 180.802} C_DIS
LIN {X -0.125,Y -403.921,Z 515.795,A 0.000,B 0.000,C 90.000,E1 179.083} C_DIS
LIN {X -0.066,Y -402.322,Z 515.774,A 0.000,B 0.000,C 90.000,E1 175.241} C_DIS
LIN {X 0.184,Y -401.895,Z 515.760,A 0.000,B 0.000,C 90.000,E1 172.761} C_DIS
LIN {X 0.074,Y -401.888,Z 515.744,A 0.000,B 0.000,C 90.000,E1 169.982} C_DIS
LIN {X 0.179,Y -402.228,Z 515.729,A 0.000,B 0.000,C 90.000,E1 167.173} C_DIS
LIN {X 0.002,Y -402.941,Z 515.715,A 0.000,B 0.000,C 90.000,E1 164.755} C_DIS
LIN {X -0.023,Y -403.650,Z 515.706,A 0.000,B 0.000,C 90.000,E1 163.015} C_DIS
LIN {X -0.104,Y -405.068,Z 515.690,A 0.000,B 0.000,C 90.000,E1 160.242} C_DIS
LIN {X 0.184,Y -406.156,Z 515.681,A 0.000,B 0.000,C 90.000,E1 158.465} C_DIS
LIN {X 0.108,Y -407.889,Z 515.667,A 0.000,B 0.000,C 90.000,E1 156.049} C_DIS
LIN {X 0.037,Y -409.865,Z 515.654,A 0.000,B 0.000,C 90.000,E1 153.640} C_DIS
LIN {X 0.178,Y -411.187,Z 515.644,A 0.000,B 0.000,C 90.000,E1 151.897} C_DIS
LIN {X -0.021,Y -412.472,Z 515.635,A 0.000,B 0.000,C 90.000,E1 150.205} C_DIS
LIN {X 0.155,Y -413.828,Z 515.623,A 0.000,B 0.000,C 90.000,E1 148.122} C_DIS
LIN {X 0.013,Y -415.093,Z 515.612,A 0.000,B 0.000,C 90.000,E1 146.087} C_DIS
LIN {X 0.023,Y -416.173,Z 515.600,A 0.000,B 0.000,C 90.000,E1 144.036} C_DIS
LIN {X -0.131,Y -417.020,Z 515.591,A 0.000,B 0.000,C 90.000,E1 142.351} C_DIS
LIN {X -0.091,Y -417.696,Z 515.581,A 0.000,B 0.000,C 90.000,E1 140.642} C_DIS
LIN {X -0.036,Y -418.285,Z 515.572,A 0.000,B 0.000,C 90.000,E1 138.933} C_DIS
LIN {X 0.106,Y -418.699,Z 515.564,A 0.000,B 0.000,C 90.000,E1 137.553} C_DIS
LIN {X -0.055,Y -418.898,Z 515.557,A 0.000,B 0.000,C 90.000,E1 136.215} C_DIS
LIN {X 0.079,Y -418.995,Z 515.549,A 0.000,B 0.000,C 90.000,E1 134.838} C_DIS
LIN {X -0.074,Y -418.929,Z 515.542,A 0.000,B 0.000,C 90.000,E1 133.500} C_DIS
